// TwinCAT 3 PLC project PLC1
// ProgramVersion: 3.1.4023.0
// libraries:
//   SPT Base Types, * (Beckhoff Automation LLC)
//   SPT Components, * (Beckhoff Automation LLC)
//   SPT Diagnostic, * (Beckhoff Automation LLC)
//   SPT EtherCat, * (Beckhoff Automation LLC)
//   SPT Event Logger, * (Beckhoff Automation LLC)
//   SPT Utilities, * (Beckhoff Automation LLC)
//   Tc2_EtherCAT, * (Beckhoff Automation GmbH)
//   Tc2_Standard, * (Beckhoff Automation GmbH)
//   Tc2_System, * (Beckhoff Automation GmbH)
//   Tc3_EventLogger, * (Beckhoff Automation GmbH)
//   Tc3_Module, * (Beckhoff Automation GmbH)
//   Tc3_PackML_V2, * (Beckhoff Automation GmbH)
//   VisuDialogs, * (System)
//   VisuSymbols,newest,System
// project tree:
//   DUTs/Recipe/NewFolder1/ ST_PullWheelsRecipe.TcDUT, ST_SealerRecipe.TcDUT, ST_UnwindRecipe.TcDUT
//   DUTs/Recipe/ ST_AxisRecipe.TcDUT, ST_ConveyorRecipe.TcDUT, ST_MotionLinxAxisRecipe.TcDUT, ST_StationRecipe.TcDUT, ST_Vision_Volume_Recipe.TcDUT, ST_Diagnostics_Recipe.TcDUT, ST_Gluer_Recipe.TcDUT, ST_DiverterRecipe.TcDUT, ST_Closer_Recipe.TcDUT, ST_LabelerRecipe.TcDUT, ST_OutfeedRecipe.TcDUT, ST_SafetyRecipe.TcDUT
//   DUTs/ ST_Descriptor2.TcDUT (not stored), ST_PackML_Control.TcDUT (not stored), ST_PackML_Control_Simplified.TcDUT (not stored)
//   / GlobalTextList.TcGTLO, MAIN.TcPOU, PlcTask.TcTTO, VisualizationManager.TcVMO (not stored)
//   Machine/Components/Contactor/ FB_Contactor.TcPOU, FB_Contactor_Dual_InOut.TcPOU, FB_Contactor_With_Dual_Feedback.TcPOU, FB_Contactor_With_Single_Feedback.TcPOU, I_Contactor.TcIO, ST_Contactor_Command.TcDUT, ST_Contactor_Config.TcDUT, ST_Contactor_HMI.TcDUT, ST_Contactor_Status.TcDUT
//   Machine/Components/Cylinder/ FB_Cylinder.TcPOU (not stored), I_Cylinder.TcIO (not stored), ST_Cylinder_Command.TcDUT (not stored), ST_Cylinder_Config.TcDUT (not stored), ST_Cylinder_HMI.TcDUT (not stored), ST_Cylinder_Status.TcDUT (not stored)
//   Machine/Components/Drives/ iDM_DriveHealth.TcIO
//   Machine/Components/Drives/Omron/ eDriveStates.TcDUT, eOmronStatus.TcDUT (not stored), FB_BLINKER_PLAY.TcPOU (not stored), FB_Omron_Inv.TcPOU, stOmronDriveMapping.TcDUT
//   Machine/Components/Drives/Omron/Old System/DM_Omron/ DM_Omron_Drive.TcPOU
//   Machine/Components/Drives/Roller Drives/2 Motor Drive/Axis/ FB_Drive_Type_1_Axis.TcPOU, I_Drive_Type_1_Axis.TcIO
//   Machine/Components/Drives/Roller Drives/2 Motor Drive/ FB_Drive_Type_1_Controller.TcPOU, I_Drive_Type_1_Controller.TcIO
//   Machine/Components/ FB_SealBar.TcPOU (not stored)
//   Machine/Components/MotionLinxAI/Axis/ FB_MotionlinxAI_Axis.TcPOU, I_MotionlinxAI_Axis.TcIO, MotionlinxAI_Error_States.TcDUT, MotionlinxAI_Motor_Status.TcDUT, ST_MotionlinxAI_Axis_Command.TcDUT, ST_MotionlinxAI_Axis_Config.TcDUT, ST_MotionlinxAI_Axis_HMI.TcDUT, ST_MotionlinxAI_Axis_Status.TcDUT
//   Machine/Components/MotionLinxAI/Axis/HMI/ ST_MotionlinxAI_Controller_Command.TcDUT, ST_MotionlinxAI_Controller_Config.TcDUT, ST_MotionlinxAI_Controller_HMI.TcDUT, ST_MotionlinxAI_Controller_Status.TcDUT
//   Machine/Components/MotionLinxAI/Controller/ FB_MotionlinxAI_Controller.TcPOU, I_MotionlinxAI_Controller_Sts.TcIO, ST_Controller_Status.TcDUT
//   Machine/Components/MotionLinxAI/ MotionlinxAI_States.TcDUT
//   Machine/Components/Relay/ I_Relay.TcIO, Relay.TcPOU, Relay_Pulse.TcPOU
//   Machine/Components/Robots/ GVL_UR.TcGVL
//   Machine/Components/Robots/UR/ fbUR.TcPOU
//   Machine/Components/Robots/UR/IO-Mapping/Structs/ stUR_EIO_Output_Mapping.TcDUT, stUR_EIO_Safety_Bits_Mapping.TcDUT, UR_Output_Data.TcDUT, UR_Safety_Bits_Data.TcDUT
//   Machine/Components/Vision/Cognex/ FB_A100.TcPOU
//   Machine/EquipmentModules/Conveyors/ FB_Robot_Outfeed_Conveyor_Module.TcPOU, FB_SingleDrive_Conveyor_With_Out_Sensor.TcPOU, FB_SingleDrive_Conveyor_With_Out_Sensor_And_Stopper.TcPOU, FB_Single_Drive_Outfeed_Sensor.TcPOU
//   Machine/EquipmentModules/ FB_Diverter_Module.TcPOU, FB_Station_Module.TcPOU, FB_Labeler_Module.TcPOU, FB_Closer_Gluer_Module.TcPOU, FB_Outfeed_Conveyor_Module_OLD.TcPOU (excluded from build)
//   Machine/EquipmentSubModules/ FB_Diverter_Module001.TcPOU, FB_Gluer_Module.TcPOU, FB_Vision_Volume_SubModule.TcPOU, FB_Vision_Barcode_SubModule.TcPOU, FB_Labeler_SubModule.TcPOU
//   Machine/ FB_Machine.TcPOU, FB_Safety.TcPOU (excluded from build), FB_Systems.TcPOU (excluded from build)
//   Machine/HMI Connections/ FB_ControlSource_HMI.TcPOU (not stored), FB_ControlSource_HMI_Machine.TcPOU
//   Machine/MachineSubModules/ FB_Diagnostics_SubModule.TcPOU, FB_Systems_Module.TcPOU
//   Machine/SafetyModules/ FB_Safety_Module.TcPOU
//   Machine/Templates/ FB_EquipmentModuleTemplate.TcPOU (not stored)
//   Machine/VISUs/VisuOjects/ V_EtherCatMasterComponent.TcVIS, V_MachineModule.TcVIS, V_SafetyModule.TcVIS, V_Module.TcVIS (not stored)
//   Machine/VISUs/ V_Main.TcVIS
// real-time tasks:
//   TASK PlcTask: cycle T#10ms, priority 10, ADS port 350
// motion (NC):
//   TASK NC-Task 1 SAF: cycle T#2ms, priority 4, ADS port 501
//   TASK NC-Task 1 SVB: cycle T#10ms, priority 8, ADS port 511
//   AXIS Unwind (id 4)
//   AXIS Seal (id 5)
//   AXIS Pull 1 (id 6)
//   AXIS Pull 2 (id 7)
// I/O:
//   DEVICE Device 2 (RT-Ethernet Adapter) DO NOT DELETE
//   DEVICE Device 5 (EtherCAT), AmsNetId 192.168.100.70.6.1
//     Box 1 (CU2508) [CU2508 Ethernet Port]
//     Term 2 (EK1100) [EK1100 EtherCAT Coupler (2A E-Bus)]
//       Term 3 (EL1904) [EL1904, 4 Ch. Safety Input 24V, TwinSAFE]
//         modules: Module 1 (FSOES)
//       Term 4 (EL1904) [EL1904, 4 Ch. Safety Input 24V, TwinSAFE]
//         modules: Module 1 (FSOES)
//       Term 5 (EL2904) [EL2904, 4 Ch. Safety Output 24V, 0.5A, TwinSAFE]
//         modules: Module 1 (FSOES), Module 2 (DO)
//       Term 6 (EL6900) [EL6900, TwinSAFE PLC]
//       Term 7 (EL2008) [EL2008 8Ch. Dig. Output 24V, 0.5A]
//       Term 8 (EL1008) [EL1008 8Ch. Dig. Input 24V, 3ms]
//       Term 9 (EL9011) [EL9011 End Terminal]
//     Box 18 (MotionLinx-Ai PLCmode) [MotionLinx-Ai PLCmode FW4.1]
// variable links:
//   PLC1/PLC1 Instance <-> Device 5 (EtherCAT)
//     PlcTask Inputs/MAIN.Machine.Systems_SubModule.Diagnostics.EtherCatMasterX001.EtherCatMaster.AmsNetID <-> InfoData/AmsNetId
//     PlcTask Inputs/MAIN.Machine.Systems_SubModule.Diagnostics.EtherCatMasterX001.EtherCatMaster.CfgSlaveCount <-> InfoData/CfgSlaveCount
//     PlcTask Inputs/MAIN.Machine.Systems_SubModule.Diagnostics.EtherCatMasterX001.EtherCatMaster.ChangeCount <-> InfoData/ChangeCount
//     PlcTask Inputs/MAIN.Machine.Systems_SubModule.Diagnostics.EtherCatMasterX001.EtherCatMaster.DevID <-> InfoData/DevId
//     PlcTask Inputs/MAIN.Machine.Systems_SubModule.Diagnostics.EtherCatMasterX001.EtherCatMaster.DevState <-> Inputs/DevState
//     PlcTask Inputs/MAIN.Machine.Systems_SubModule.Diagnostics.EtherCatMasterX001.EtherCatMaster.SlaveCount <-> Inputs/SlaveCount
//     PlcTask Inputs/MAIN.Machine.Systems_SubModule.Diagnostics.EtherCatMasterX001.FrmXWcState[0] <-> Inputs/Frm0State
//   PLC1/PLC1 Instance <-> Device 5 (EtherCAT)/Box 18 (MotionLinx-Ai PLCmode)
//     PlcTask Inputs/MAIN.Machine.Diverter_MotionlinxAI_Controller.bInputToggle <-> WcState/InputToggle
//     PlcTask Inputs/MAIN.Machine.Diverter_MotionlinxAI_Controller.bWCState <-> WcState/WcState
//     PlcTask Inputs/MAIN.Machine.Diverter_MotionlinxAI_Controller.iSensors <-> Module Inputs/AllSensors
//     PlcTask Inputs/MAIN.Machine.Diverter_MotionlinxAI_Controller.iSysDiagnostics <-> Module Diagnostics/SystemDiagnostic
//     PlcTask Inputs/MAIN.Machine.Station_1.Axis.iDiagnostics <-> Module Diagnostics/DiagnosticLeft
//     PlcTask Inputs/MAIN.Machine.Station_1.Axis.iPosition <-> Module Inputs/PositionLeft
//     PlcTask Inputs/MAIN.Machine.Station_1.Axis.iServoState <-> Module Inputs/ServoStateL
//     PlcTask Inputs/MAIN.Machine.Station_5.Axis.iDiagnostics <-> Module Diagnostics/DiagnosticRight
//     PlcTask Inputs/MAIN.Machine.Station_5.Axis.iPosition <-> Module Inputs/PositionRight
//     PlcTask Inputs/MAIN.Machine.Station_5.Axis.iServoState <-> Module Inputs/ServoStateR
//     PlcTask Outputs/MAIN.Machine.Diverter_MotionlinxAI_Controller.oClearMotorError <-> Servo/Periphery/ClearMotorError
//     PlcTask Outputs/MAIN.Machine.Diverter_MotionlinxAI_Controller.oServoControl <-> Servo/Periphery/ServoCtrl
//     PlcTask Outputs/MAIN.Machine.Diverter_MotionlinxAI_Controller.oSetPin2Out <-> Servo/Periphery/WritePin2Output
//     PlcTask Outputs/MAIN.Machine.Station_1.Axis.oMotorAccel <-> Motor Ramps/AccelLeft
//     PlcTask Outputs/MAIN.Machine.Station_1.Axis.oMotorBrakeMode <-> Motor Setup/BrakeModeLeft
//     PlcTask Outputs/MAIN.Machine.Station_1.Axis.oMotorControl <-> Motor Setup/MDRCtrlLeft
//     PlcTask Outputs/MAIN.Machine.Station_1.Axis.oMotorDecel <-> Motor Ramps/DecelLeft
//     PlcTask Outputs/MAIN.Machine.Station_1.Axis.oMotorSpeed <-> Motor Setup/SpeedLeft
//     PlcTask Outputs/MAIN.Machine.Station_1.Axis.oServoPos <-> Servo/Periphery/ServoLeft
//     PlcTask Outputs/MAIN.Machine.Station_5.Axis.oMotorAccel <-> Motor Ramps/AccelRight
//     PlcTask Outputs/MAIN.Machine.Station_5.Axis.oMotorBrakeMode <-> Motor Setup/BrakeModeRight
//     PlcTask Outputs/MAIN.Machine.Station_5.Axis.oMotorControl <-> Motor Setup/MDRCtrlRight
//     PlcTask Outputs/MAIN.Machine.Station_5.Axis.oMotorDecel <-> Motor Ramps/DecelRight
//     PlcTask Outputs/MAIN.Machine.Station_5.Axis.oMotorSpeed <-> Motor Setup/SpeedRight
//     PlcTask Outputs/MAIN.Machine.Station_5.Axis.oServoPos <-> Servo/Periphery/ServoRight
//   PLC1/PLC1 Instance <-> Device 5 (EtherCAT)/Term 2 (EK1100)/Term 6 (EL6900)
//     PlcTask Inputs/MAIN.Machine.Safety_SubModule.SafetyEstop.InfoData/Diag <-> TwinSAFE Group Info Data/TwinSafeGroup_Estop Info Data/Diag
//     PlcTask Inputs/MAIN.Machine.Safety_SubModule.SafetyEstop.InfoData/State <-> TwinSAFE Group Info Data/TwinSafeGroup_Estop Info Data/State
//     PlcTask Inputs/MAIN.Machine.Safety_SubModule.SafetyGroup_ESTOP.InfoData/Diag <-> Function Block Info Data/TwinSafeGroup_Estop.ESTOP_Circuit.FBEstop1 Info Data/Diag
//     PlcTask Inputs/MAIN.Machine.Safety_SubModule.SafetyGroup_ESTOP.InfoData/State <-> Function Block Info Data/TwinSafeGroup_Estop.ESTOP_Circuit.FBEstop1 Info Data/State
//     PlcTask Inputs/MAIN.Machine.Safety_SubModule.SafetyGroup_IO.InfoData/Diag <-> TwinSAFE Group Info Data/TwinSafeGroup_IO Info Data/Diag
//     PlcTask Inputs/MAIN.Machine.Safety_SubModule.SafetyGroup_IO.InfoData/State <-> TwinSAFE Group Info Data/TwinSafeGroup_IO Info Data/State
//     PlcTask Inputs/MAIN.Machine.Safety_SubModule.SafetyInput.InfoData/Diag <-> Connection Info Data/Message_5 Info Data/Diag
//     PlcTask Inputs/MAIN.Machine.Safety_SubModule.SafetyInput.InfoData/State <-> Connection Info Data/Message_5 Info Data/State
//     PlcTask Inputs/MAIN.Machine.Safety_SubModule.SafetyOutput.InfoData/Diag <-> Connection Info Data/Message_7 Info Data/Diag
//     PlcTask Inputs/MAIN.Machine.Safety_SubModule.SafetyOutput.InfoData/State <-> Connection Info Data/Message_7 Info Data/State
//     PlcTask Outputs/MAIN.Machine.Safety_SubModule.SafetyGroup_ESTOP.Run <-> StandardOutputs/Standard In Var 14
//     PlcTask Outputs/MAIN.Machine.Safety_SubModule.SafetyGroup_IO.Run <-> StandardOutputs/Standard In Var 4
//     PlcTask Outputs/MAIN.Machine.Safety_SubModule.Safty_Reset_Pulse_Out.output <-> StandardOutputs/Standard In Var 12
//     PlcTask Outputs/MAIN.Machine.Safety_SubModule.Safty_Reset_Pulse_Out.output <-> StandardOutputs/Standard In Var 3
//   (this object) <-> Device 5 (EtherCAT)
//     Term 2 (EK1100)/Term 3 (EL1904)/Module 1 (FSOES)/RxPDO/FSOE <-> Term 2 (EK1100)/Term 6 (EL6900)/ConnectionInputs/Message_5 TxPDO
//     Term 2 (EK1100)/Term 5 (EL2904)/Module 1 (FSOES)/RxPDO/FSOE <-> Term 2 (EK1100)/Term 6 (EL6900)/ConnectionInputs/Message_7 TxPDO
//     Term 2 (EK1100)/Term 3 (EL1904)/Module 1 (FSOES)/TxPDO/FSOE <-> Term 2 (EK1100)/Term 6 (EL6900)/ConnectionOutputs/Message_5 RxPDO
//     Term 2 (EK1100)/Term 5 (EL2904)/Module 1 (FSOES)/TxPDO/FSOE <-> Term 2 (EK1100)/Term 6 (EL6900)/ConnectionOutputs/Message_7 RxPDO
//     Term 2 (EK1100)/Term 6 (EL6900)/ConnectionInputs/Message_5 TxPDO <-> Term 2 (EK1100)/Term 3 (EL1904)/Module 1 (FSOES)/RxPDO/FSOE
//     Term 2 (EK1100)/Term 6 (EL6900)/ConnectionInputs/Message_7 TxPDO <-> Term 2 (EK1100)/Term 5 (EL2904)/Module 1 (FSOES)/RxPDO/FSOE
//     Term 2 (EK1100)/Term 6 (EL6900)/ConnectionOutputs/Message_5 RxPDO <-> Term 2 (EK1100)/Term 3 (EL1904)/Module 1 (FSOES)/TxPDO/FSOE
//     Term 2 (EK1100)/Term 6 (EL6900)/ConnectionOutputs/Message_7 RxPDO <-> Term 2 (EK1100)/Term 5 (EL2904)/Module 1 (FSOES)/TxPDO/FSOE

CONFIGURATION PLC1
    RESOURCE PLC ON TwinCAT3
        TASK PlcTask(INTERVAL := T#10ms, PRIORITY := 10);
        PROGRAM MAIN WITH PlcTask : MAIN;
    END_RESOURCE
END_CONFIGURATION

// ---- DUTs/Recipe/NewFolder1/ST_PullWheelsRecipe.TcDUT
TYPE ST_PullWheelsRecipe :
	STRUCT
		Length				: LREAL;
		LeftAxis			: ST_AxisRecipe;
		RightAxis			: ST_AxisRecipe;
		CylinderExtendTime	: LREAL;
		CylinderRetractTime : LREAL;
	END_STRUCT
END_TYPE

// ---- DUTs/Recipe/NewFolder1/ST_SealerRecipe.TcDUT
TYPE ST_SealerRecipe :
	STRUCT
		Axis		   : ST_AxisRecipe;
		Temp		   : LREAL;
		SealTime	   : LREAL;
		OpenPosition   : LREAL;
		ClosedPosition : LREAL;
	END_STRUCT
END_TYPE

// ---- DUTs/Recipe/NewFolder1/ST_UnwindRecipe.TcDUT
TYPE ST_UnwindRecipe :
	STRUCT
		Axis : ST_AxisRecipe;
	END_STRUCT
END_TYPE

// ---- DUTs/Recipe/ST_AxisRecipe.TcDUT
TYPE ST_AxisRecipe :
	STRUCT
		Velocity		: INT;
		Acceleration	: INT;
		Deceleration	: INT;
	//	Speed			: INT;
		MaxVelocity		: INT;
	END_STRUCT
END_TYPE

// ---- DUTs/Recipe/ST_ConveyorRecipe.TcDUT
TYPE ST_ConveyorRecipe :
	STRUCT
		Axis : ST_MotionLinxAxisRecipe;
		
	END_STRUCT
END_TYPE

// ---- DUTs/Recipe/ST_MotionLinxAxisRecipe.TcDUT
TYPE ST_MotionLinxAxisRecipe :
	STRUCT
		Velocity		: INT;
		Acceleration	: INT;
		Deceleration	: INT;	
		MaxSpeed		:UINT;
	END_STRUCT
END_TYPE

// ---- DUTs/Recipe/ST_StationRecipe.TcDUT
TYPE ST_StationRecipe :
STRUCT

		Axis			: ST_AxisRecipe;
		//	Travel Time ??
END_STRUCT
END_TYPE

// ---- DUTs/Recipe/ST_Vision_Volume_Recipe.TcDUT
TYPE ST_Vision_Volume_Recipe :
	STRUCT
		Length				: LREAL;
//		LeftAxis			: ST_AxisRecipe;
//		RightAxis			: ST_AxisRecipe;
		CylinderExtendTime	: LREAL;
		CylinderRetractTime : LREAL;
	END_STRUCT
END_TYPE

// ---- DUTs/Recipe/ST_Diagnostics_Recipe.TcDUT
TYPE ST_Diagnostics_Recipe :
	STRUCT
		Length				: LREAL;
//		LeftAxis			: ST_AxisRecipe;
//		RightAxis			: ST_AxisRecipe;
		CylinderExtendTime	: LREAL;
		CylinderRetractTime : LREAL;
	END_STRUCT
END_TYPE

// ---- DUTs/Recipe/ST_Gluer_Recipe.TcDUT
TYPE ST_Gluer_Recipe :
	STRUCT
		Length				: LREAL;
			// Data
		SetTemperature	   : LREAL;
		Trigger_Delay		: TIME;	
//		LeftAxis			: ST_AxisRecipe;
//		RightAxis			: ST_AxisRecipe;
		CylinderExtendTime	: LREAL;
		CylinderRetractTime : LREAL;
	END_STRUCT
END_TYPE

// ---- DUTs/Recipe/ST_DiverterRecipe.TcDUT
TYPE ST_DiverterRecipe :
	STRUCT
		Length				: LREAL;
//		LeftAxis			: ST_AxisRecipe;
//		RightAxis			: ST_AxisRecipe;
		CylinderExtendTime	: LREAL;
		CylinderRetractTime : LREAL;
	END_STRUCT
END_TYPE

// ---- DUTs/Recipe/ST_Closer_Recipe.TcDUT
TYPE ST_Closer_Recipe :
	STRUCT
		Length				: LREAL;
//		LeftAxis			: ST_AxisRecipe;
//		RightAxis			: ST_AxisRecipe;
		CylinderExtendTime	: LREAL;
		CylinderRetractTime : LREAL;
	END_STRUCT
END_TYPE

// ---- DUTs/Recipe/ST_LabelerRecipe.TcDUT
TYPE ST_LabelerRecipe :
	STRUCT
		Length				: LREAL;
//		LeftAxis			: ST_AxisRecipe;
//		RightAxis			: ST_AxisRecipe;
		CylinderExtendTime	: LREAL;
		CylinderRetractTime : LREAL;
	END_STRUCT
END_TYPE

// ---- DUTs/Recipe/ST_OutfeedRecipe.TcDUT
TYPE ST_OutfeedRecipe :
	STRUCT
		Length				: LREAL;
//		LeftAxis			: ST_AxisRecipe;
//		RightAxis			: ST_AxisRecipe;
		CylinderExtendTime	: LREAL;
		CylinderRetractTime : LREAL;
	END_STRUCT
END_TYPE

// ---- DUTs/Recipe/ST_SafetyRecipe.TcDUT
TYPE ST_SafetyRecipe :
	STRUCT
		Axis : ST_AxisRecipe;
	END_STRUCT
END_TYPE

// ---- Machine/Components/Contactor/ST_Contactor_Command.TcDUT
TYPE ST_Contactor_Command :
    STRUCT
        Extend  : BOOL;
        Retract : BOOL;
    END_STRUCT
END_TYPE

// ---- Machine/Components/Contactor/ST_Contactor_Config.TcDUT
TYPE ST_Contactor_Config :
    STRUCT
        ExtendTime  : LREAL;
        RetractTime : LREAL;
    END_STRUCT
END_TYPE

// ---- Machine/Components/Contactor/ST_Contactor_HMI.TcDUT
TYPE ST_Contactor_HMI :
    STRUCT
        Config  : ST_Contactor_Config;
        Command : ST_Contactor_Command;
        Status  : ST_Contactor_Status;
    END_STRUCT
END_TYPE

// ---- Machine/Components/Contactor/ST_Contactor_Status.TcDUT
TYPE ST_Contactor_Status :
    STRUCT
        Extended   : BOOL;
        Retracted  : BOOL;
        Extending  : BOOL;
        Retracting : BOOL;
    END_STRUCT
END_TYPE

// ---- Machine/Components/Drives/Omron/eDriveStates.TcDUT
{attribute 'qualified_only'}
{attribute 'strict'}
{attribute 'to_string'}
TYPE eDriveStates :
(
	FAULT := 0,
	FAULT_STOPPING,
 	AWAITING_RESET,
	RESET,
	DISABLED,
	STOPPED,	
	STOPPING,
	STARTING,
	RUNNING
);
END_TYPE

// ---- Machine/Components/Drives/Omron/stOmronDriveMapping.TcDUT
TYPE stOmronDriveMapping :
STRUCT
	
	//Inputs
	inInputTerminal AT %I* : UINT;
	inMotorCurrent AT %I* : UINT;	
	inFinTemp AT %I* : UINT;
	inStatus AT %I* : UINT;
	inOutputFrequency AT %I* : UINT;	
	ibWcState AT %I* : BOOL;
	
	inPulse AT %I* : UINT; // not used 

	inErrorCode AT %I* : UINT;  // NOT used 
	inErrorSubCode AT %I* : UINT; // not used 
	inSTOActive  	AT %I* : BOOL; // not mapped 
		
	//Outputs
	onCommand AT %Q* : UINT;
	onFrequencyRef AT %Q* : UINT;
	onAccelTime AT %Q* : UINT;
	onDecelTime AT %Q* : UINT;
			
END_STRUCT
END_TYPE

// ---- Machine/Components/MotionLinxAI/Axis/HMI/ST_MotionlinxAI_Controller_Command.TcDUT
TYPE ST_MotionlinxAI_Controller_Command :
	STRUCT
		Extend	: BOOL;
		Retract : BOOL;
	END_STRUCT
END_TYPE

// ---- Machine/Components/MotionLinxAI/Axis/HMI/ST_MotionlinxAI_Controller_Config.TcDUT
TYPE ST_MotionlinxAI_Controller_Config :
	STRUCT
		ExtendTime	: LREAL;
		RetractTime : LREAL;
	END_STRUCT
END_TYPE

// ---- Machine/Components/MotionLinxAI/Axis/HMI/ST_MotionlinxAI_Controller_HMI.TcDUT
TYPE ST_MotionlinxAI_Controller_HMI :
	STRUCT
		Config	: ST_MotionlinxAI_Controller_Config;
		Command : ST_MotionlinxAI_Controller_Command;
		Status	: ST_MotionlinxAI_Controller_Status;
	END_STRUCT
END_TYPE

// ---- Machine/Components/MotionLinxAI/Axis/HMI/ST_MotionlinxAI_Controller_Status.TcDUT
TYPE ST_MotionlinxAI_Controller_Status :
	STRUCT
		Extended   : BOOL;
		Retracted  : BOOL;
		Extending  : BOOL;
		Retracting : BOOL;
	END_STRUCT
END_TYPE

// ---- Machine/Components/MotionLinxAI/Axis/MotionlinxAI_Error_States.TcDUT
{attribute 'qualified_only'}
{attribute 'strict'}
TYPE MotionlinxAI_Error_States :
(
	
	NO_ERROR,
	MOTOR_SPEED_HI,
	MOTOR_SPEED_LO,
	MOTOR_BOARD_OVERHEAT,
	MOTOR_OVERVOLTAGE,
	MOTOR_UNDERVOLTAGE,
	MOTOR_OVERHEATED,
	MOTOR_MAX_TORQUE,
	MOTOR_SHORT_CIRCUIT,
	MOTOR_NOT_CONNECTED,
	MOTOR_OVERLOADED,
	MOTOR_STALLED,
	MOTOR_HALL_SENSOR
);
END_TYPE

// ---- Machine/Components/MotionLinxAI/Axis/MotionlinxAI_Motor_Status.TcDUT
{attribute 'qualified_only'}
TYPE MotionlinxAI_Motor_Status :
(
	MOTOR_NOT_RUNNING_BRAKED := 0 ,
	MOTOR_NOT_RUNNING_UNBRAKED,
	MOTOR_RUNNING_CCW,
	MOTOR_RUNNING_CW

);
END_TYPE

// ---- Machine/Components/MotionLinxAI/Axis/ST_MotionlinxAI_Axis_Command.TcDUT
TYPE ST_MotionlinxAI_Axis_Command :
	STRUCT
		Extend	: BOOL;
		Retract : BOOL;
	END_STRUCT
END_TYPE

// ---- Machine/Components/MotionLinxAI/Axis/ST_MotionlinxAI_Axis_Config.TcDUT
TYPE ST_MotionlinxAI_Axis_Config :
	STRUCT
		ExtendTime	: LREAL;
		RetractTime : LREAL;
	END_STRUCT
END_TYPE

// ---- Machine/Components/MotionLinxAI/Axis/ST_MotionlinxAI_Axis_HMI.TcDUT
TYPE ST_MotionlinxAI_Axis_HMI :
	STRUCT
		Config	: ST_MotionlinxAI_Axis_Config;
		Command : ST_MotionlinxAI_Axis_Command;
		Status	: ST_MotionlinxAI_Axis_Status;
	END_STRUCT
END_TYPE

// ---- Machine/Components/MotionLinxAI/Axis/ST_MotionlinxAI_Axis_Status.TcDUT
TYPE ST_MotionlinxAI_Axis_Status :
	STRUCT
		Extended   : BOOL;
		Retracted  : BOOL;
		Extending  : BOOL;
		Retracting : BOOL;
	END_STRUCT
END_TYPE

// ---- Machine/Components/MotionLinxAI/Controller/ST_Controller_Status.TcDUT
TYPE ST_Controller_Status :
STRUCT
	HasFault : BOOL;
	bEnabled : BOOL;
	Sensors : INT;
END_STRUCT
END_TYPE

// ---- Machine/Components/MotionLinxAI/MotionlinxAI_States.TcDUT
{attribute 'qualified_only'}
{attribute 'strict'}
TYPE MotionlinxAI_States :
(
	ERROR := 0,
	HOMING,
	STOPPED,
	RUNNING
);
END_TYPE

// ---- Machine/Components/Robots/UR/IO-Mapping/Structs/stUR_EIO_Output_Mapping.TcDUT
TYPE stUR_EIO_Output_Mapping :
STRUCT
	obBrakeRelease		:	BIT;
	{attribute 'hide'}
	Reserved_UR_1  : BIT;
	{attribute 'hide'}
	Reserved_UR_2  : BIT;
	{attribute 'hide'}
	Reserved_UR_3  : BIT;
	{attribute 'hide'}
	Reserved_UR_4  : BIT;
	{attribute 'hide'}
	Reserved_UR_5  : BIT;
	{attribute 'hide'}
	Reserved_UR_6  : BIT;
	{attribute 'hide'}
	Reserved_UR_7  : BIT;
	{attribute 'hide'}
	Reserved_UR_8  : BIT;
	{attribute 'hide'}
	Reserved_UR_9  : BIT;
	{attribute 'hide'}
	Reserved_UR_10  : BIT;
	{attribute 'hide'}
	Reserved_UR_11  : BIT;
	{attribute 'hide'}
	Reserved_UR_12  : BIT;
	{attribute 'hide'}
	Reserved_UR_13  : BIT;
	{attribute 'hide'}
	Reserved_UR_14  : BIT;
	{attribute 'hide'}
	Reserved_UR_15  : BIT;
	{attribute 'hide'}
	Reserved_UR_16  : BIT;
	{attribute 'hide'}
	Reserved_UR_17  : BIT;
	{attribute 'hide'}
	Reserved_UR_18  : BIT;
	{attribute 'hide'}
	Reserved_UR_19  : BIT;
	{attribute 'hide'}
	Reserved_UR_20  : BIT;
	{attribute 'hide'}
	Reserved_UR_21  : BIT;
	{attribute 'hide'}
	Reserved_UR_22  : BIT;
	{attribute 'hide'}
	Reserved_UR_23  : BIT;
	{attribute 'hide'}
	Reserved_UR_24  : BIT;
	{attribute 'hide'}
	Reserved_UR_25  : BIT;
	{attribute 'hide'}
	Reserved_UR_26  : BIT;
	{attribute 'hide'}
	Reserved_UR_27  : BIT;
	{attribute 'hide'}
	Reserved_UR_28  : BIT;
	{attribute 'hide'}
	Reserved_UR_29  : BIT;
	{attribute 'hide'}
	Reserved_UR_30  : BIT;
	{attribute 'hide'}
	Reserved_UR_31  : BIT;
END_STRUCT
END_TYPE

// ---- Machine/Components/Robots/UR/IO-Mapping/Structs/stUR_EIO_Safety_Bits_Mapping.TcDUT
TYPE stUR_EIO_Safety_Bits_Mapping :
STRUCT
	ibNormalMode   : BIT;
	ibReducedMode  : BIT;
	{attribute 'hide'}
	Reserved_UR_2  : BIT;
	{attribute 'hide'}
	Reserved_UR_3  : BIT;
	{attribute 'hide'}
	Reserved_UR_4  : BIT;
	{attribute 'hide'}
	Reserved_UR_5  : BIT;
	{attribute 'hide'}
	Reserved_UR_6  : BIT;
	{attribute 'hide'}
	Reserved_UR_7  : BIT;
	{attribute 'hide'}
	Reserved_UR_8  : BIT;
	{attribute 'hide'}
	Reserved_UR_9  : BIT;
	{attribute 'hide'}
	Reserved_UR_10  : BIT;
	{attribute 'hide'}
	Reserved_UR_11  : BIT;
	{attribute 'hide'}
	Reserved_UR_12  : BIT;
	{attribute 'hide'}
	Reserved_UR_13  : BIT;
	{attribute 'hide'}
	Reserved_UR_14  : BIT;
	{attribute 'hide'}
	Reserved_UR_15  : BIT;
	{attribute 'hide'}
	Reserved_UR_16  : BIT;
	{attribute 'hide'}
	Reserved_UR_17  : BIT;
	{attribute 'hide'}
	Reserved_UR_18  : BIT;
	{attribute 'hide'}
	Reserved_UR_19  : BIT;
	{attribute 'hide'}
	Reserved_UR_20  : BIT;
	{attribute 'hide'}
	Reserved_UR_21  : BIT;
	{attribute 'hide'}
	Reserved_UR_22  : BIT;
	{attribute 'hide'}
	Reserved_UR_23  : BIT;
	{attribute 'hide'}
	Reserved_UR_24  : BIT;
	{attribute 'hide'}
	Reserved_UR_25  : BIT;
	{attribute 'hide'}
	Reserved_UR_26  : BIT;
	{attribute 'hide'}
	Reserved_UR_27  : BIT;
	{attribute 'hide'}
	Reserved_UR_28  : BIT;
	{attribute 'hide'}
	Reserved_UR_29  : BIT;
	{attribute 'hide'}
	Reserved_UR_30  : BIT;
	{attribute 'hide'}
	Reserved_UR_31  : BIT;

END_STRUCT
END_TYPE

// ---- Machine/Components/Robots/UR/IO-Mapping/Structs/UR_Output_Data.TcDUT
TYPE UR_Output_Data :
UNION
	odwURRawOutputData : DWORD;
	data : stUR_EIO_Output_Mapping;
END_UNION
END_TYPE

// ---- Machine/Components/Robots/UR/IO-Mapping/Structs/UR_Safety_Bits_Data.TcDUT
TYPE UR_Safety_Bits_Data :
UNION
	idwURRawInputData : DWORD;
	data : stUR_EIO_Safety_Bits_Mapping;
END_UNION
END_TYPE

// ---- Machine/Components/Robots/GVL_UR.TcGVL
{attribute 'qualified_only'}
VAR_GLOBAL
	UR		 : fbUR;

	ibURPowered				AT %I* : BOOL;
	obURPowerOn				AT %Q* : BOOL;
	
	ibURProtectiveStopOK		AT %I* : BOOL;

END_VAR

// ---- Machine/Components/Contactor/I_Contactor.TcIO
INTERFACE I_Contactor

METHOD Extend
VAR_INPUT
END_VAR
END_METHOD

PROPERTY Extended : BOOL
GET
END_GET
END_PROPERTY

PROPERTY ExtendTime : LREAL
GET
END_GET
SET
END_SET
END_PROPERTY

METHOD Retract
VAR_INPUT
END_VAR
END_METHOD

PROPERTY Retracted : BOOL
GET
END_GET
END_PROPERTY

PROPERTY RetractTime : LREAL
GET
END_GET
SET
END_SET
END_PROPERTY

END_INTERFACE

// ---- Machine/Components/Drives/iDM_DriveHealth.TcIO
INTERFACE iDM_DriveHealth

METHOD Disable : BOOL
VAR_INPUT
END_VAR
END_METHOD

METHOD Enable : BOOL
VAR_INPUT
END_VAR
END_METHOD

PROPERTY FaultLocation : STRING(50)
GET
END_GET
END_PROPERTY

PROPERTY HasFault : BOOL
GET
END_GET
END_PROPERTY

PROPERTY IsReady : BOOL
GET
END_GET
END_PROPERTY

PROPERTY IsRunning : BOOL
GET
END_GET
END_PROPERTY

METHOD Reset : BOOL
VAR_INPUT
END_VAR
END_METHOD

END_INTERFACE

// ---- Machine/Components/Drives/Roller Drives/2 Motor Drive/Axis/I_Drive_Type_1_Axis.TcIO
INTERFACE I_Drive_Type_1_Axis

METHOD Drive : BOOL
VAR_INPUT
END_VAR
END_METHOD

PROPERTY Position : real
GET
END_GET
SET
END_SET
END_PROPERTY

END_INTERFACE

// ---- Machine/Components/Drives/Roller Drives/2 Motor Drive/I_Drive_Type_1_Controller.TcIO
INTERFACE I_Drive_Type_1_Controller

END_INTERFACE

// ---- Machine/Components/MotionLinxAI/Axis/I_MotionlinxAI_Axis.TcIO
INTERFACE I_MotionlinxAI_Axis

PROPERTY HasFault : BOOL
GET
END_GET
END_PROPERTY

PROPERTY IsEnabled : BOOL
GET
END_GET
END_PROPERTY

PROPERTY IsReady : BOOL
GET
END_GET
END_PROPERTY

END_INTERFACE

// ---- Machine/Components/MotionLinxAI/Controller/I_MotionlinxAI_Controller_Sts.TcIO
INTERFACE I_MotionlinxAI_Controller_Sts

METHOD Disable : BOOL
(*BRAKING MODES:
	0 : NORMAL - HOLDS IN PLACE BY SHORTING WINDINGS
	1 : FREE - NOT HELD IN PLACE
	2 : SERVO - MAINTAINS POSITION BASED ON HALLS EFFECT SENSOR*)
END_METHOD

PROPERTY HasFault : BOOL
GET
END_GET
END_PROPERTY

PROPERTY Sensors : int
GET
END_GET
END_PROPERTY

END_INTERFACE

// ---- Machine/Components/Relay/I_Relay.TcIO
INTERFACE I_Relay

PROPERTY OFF : BOOL
GET
END_GET
END_PROPERTY

PROPERTY ON : Bool
GET
END_GET
END_PROPERTY

METHOD PUBLIC SwitchOff
VAR_INPUT
END_VAR
END_METHOD

METHOD PUBLIC SwitchOn
VAR_INPUT
END_VAR
END_METHOD

END_INTERFACE

// ---- MAIN.TcPOU
PROGRAM MAIN
VAR
	ControlSource_HMI : FB_ControlSource_HMI_Machine;
	
//	Safety		: FB_Safety			:= (Name := 'Safety', DisableSubModuleModeChange	:= TRUE, LogStateChanges	:= TRUE );
//	Systems	  	: FB_Systems := (Name := 'Machine Systems');
	Machine		: FB_Machine := (Name := 'Box Closer Labeler');
	InitComplete	  : BOOL;

	//Debug testing Recipe manager
	Value1 : INT;
	Value2 : INT;
END_VAR

CyclicLogic();
//Did you update??

METHOD CyclicLogic
VAR_INPUT
END_VAR
IF NOT InitComplete THEN
	InitComplete := Initialize();
	RETURN;
END_IF

//Machine support HMI & Production Monitor
ControlSource_HMI.CyclicLogic();

//Safety
//Safety.CyclicLogic();

//Machine Systems 	- Communications, maintenance
//Systems.CyclicLogic();


//Machine Cyclic Logic
Machine.CyclicLogic();
END_METHOD

METHOD Initialize : BOOL
VAR_INPUT
END_VAR
//Top level machine initialization should happen here, in the main initialization method. Each subsequent "layer" of modules will be named within their respective "parent" intialize method
_AppInfo.KeepOutputsOnBP := TRUE;
IF NOT ControlSource_HMI.Registered THEN
	Machine.RegisterExternalController(ControlSource_HMI);
END_IF

ControlSource_HMI.CyclicLogic();
Initialize := TRUE;
END_METHOD

END_PROGRAM

// ---- Machine/HMI Connections/FB_ControlSource_HMI_Machine.TcPOU
FUNCTION_BLOCK FB_ControlSource_HMI_Machine EXTENDS FB_ControlSource_HMI
VAR_INPUT
END_VAR

VAR_OUTPUT
END_VAR

VAR
END_VAR

METHOD CyclicLogic
VAR_INPUT
END_VAR
SUPER^.CyclicLogic();

//Change the start permissive for the Machine 
MainPMLControl_Simplified.StartPermissive := MainPMLControl_Standard.CurrentState = Tc3_PackML_V2.E_PMLState.ePMLState_Idle OR (MainPMLControl_Standard.CurrentState = Tc3_PackML_V2.E_PMLState.ePMLState_Held AND MAIN.Machine.Station_1.CurrentState = E_PMLState.ePMLState_Idle);
//MainPMLControl_Simplified.StartPermissive := MainPMLControl_Standard.CurrentState = Tc3_PackML_V2.E_PMLState.ePMLState_Idle OR (MainPMLControl_Standard.CurrentState = Tc3_PackML_V2.E_PMLState.ePMLState_Held AND MAIN.VFFSDemo.Unwind.CurrentState = E_PMLState.ePMLState_Idle);
END_METHOD

END_FUNCTION_BLOCK

// ---- Machine/FB_Machine.TcPOU
FUNCTION_BLOCK FB_Machine EXTENDS FB_PackML_BaseModule // IMPLEMENTS I_ControlsProductionRate
VAR
	
//	//FB Called  for this machine
//	Diverter_Controller_1	:FB_Drive_Type_1_Controller := (Name := 'Diverter_Controller_1');

	// Components
//	Buffer_1_Outfeed_Sensor :FB_DigitalSensor		:= (Name := 'Sensor', DebounceMode := E_DebounceMode.SimpleFlickerFilter, DebounceTime := T#250MS, Inverted    := FALSE, SimulationInput:= FALSE, SimulationMode := E_SensorSimulationMode.InputDriven) ;
	
	// Sub Modules
	//Safety
	Safety_SubModule			: FB_Safety_Module			:= (Name := 'Safety', LogStateChanges := TRUE);
	
	//Systems
	Systems_SubModule			: FB_Systems_Module	:= (Name := 'Systems', LogStateChanges := TRUE);

	
	Station_1		: FB_Station_Module:= (Name := 'Product Infeed', LogStateChanges := TRUE);
	Station_2		: FB_Station_Module:= (Name := 'Station_2', LogStateChanges := TRUE);
	Station_3		: FB_Station_Module:= (Name := 'Station_3', LogStateChanges := TRUE);
	Station_4		: FB_Station_Module:= (Name := 'Station_4', LogStateChanges := TRUE);
	Station_5			: FB_Station_Module:= (Name := 'Robot Outfeed Station', LogStateChanges := TRUE);
	Station_6		: FB_Station_Module:= (Name := 'UR Robot Station', LogStateChanges := TRUE);
//	Outfeed			: FB_Robot_Outfeed_Conveyor_Module:= (Name := 'Robot Outfeed Station', LogStateChanges := TRUE);
	

	//Initial List of Components
	ipComponents_Init : ARRAY[1..Parameters_PackML_Base.MAX_NO_OF_COMPONENTS] OF I_ComponentBase := [];
	
	//FB Called  for this machine
	Diverter_MotionlinxAI_Controller	:FB_MotionlinxAI_Controller	:= (Name := 'Diverter Drives');
	Diverter_MotionlinxAI_Controller_Sensors	: I_MotionlinxAI_Controller_Sts;
	

	//Alarms for this module
	MachineAlarms : ARRAY[1..MACHINE_ALARM_COUNT] OF FB_TcAlarm;

	//Current Recipe Name
	CurrentRecipeName : STRING;

	//Get Data From PackML? Else RecipeManager is running
	DataFromPackML : BOOL := TRUE;
	Externam_Machine	:I_PackML_ExternalController;

	//Data 
	sealTimeStart : ULINT;
	sealTimeEnd	  : ULINT;
	sealingTime	  : LREAL;
	sealTrig	  : R_TRIG;
	pullTimeStart : ULINT;
	pullTimeEnd	  : ULINT;
	pullingTime	  : LREAL;
	pulltrig	  : R_TRIG;
	partTimeStart : ULINT;
	partTimeEnd	  : ULINT;
	partTime	  : LREAL;
	parts		  : DINT;
	product		  : DINT;

	//Pack Tags for System
	{attribute 'OPC.UA.DA' := '1'}
	_PackTags : ST_PackMLv30Ext; //ST_PackMLv30 is obsolete in Tc3_PackML_V2
END_VAR

VAR CONSTANT
	//PackTag parameter IDs
	LENGTH		   : INT := 1;
	SEALTEMP	   : INT := 2;
	SEALTIME	   : INT := 3;
	PULLWHEELS_VEL : INT := 4;
	PULLWHEELS_ACC : INT := 5;
	SEALER_VEL	   : INT := 6;
	SEALER_ACC	   : INT := 7;
	UNWIND_VEL	   : INT := 8;
	UNWIND_ACC	   : INT := 9;
	OPEN_POS	   : INT := 10;
	CLOSED_POS	   : INT := 11;

	//Alarm count constant
	MACHINE_ALARM_COUNT : INT := 6;
END_VAR

// Simulation variables
VAR
	EstopInput	: BOOL;
	LowAirInput : BOOL;
	ErrorInput	: BOOL;
	WarnInput	: BOOL;
	InfoInput	: BOOL;
END_VAR

(*







*)

METHOD PROTECTED Completing
VAR_INPUT
END_VAR
CASE _CurrentMode OF
	//=================================PRODUCTION MODE==================================
	E_PMLUnitMode.ePMLUnitMode_Production:
		StateComplete();

	E_PMLUnitMode.ePMLUnitMode_Maintenance, E_PMLUnitMode.ePMLUnitMode_Manual:
		SUPER^.Completing();
END_CASE
END_METHOD

METHOD PROTECTED CreateEvents
VAR_INPUT
END_VAR
// Add your event creation here
F_CreateAllEventsInClass(Alarms		:= MachineAlarms,
						 ClassSize	:= SIZEOF(TC_Events.DemoSystem),
						 pInitEvent := ADR(TC_EVENTS.DemoSystem.InitReferenceEvent),
						 Prefix		:= Name);

// Super call to base
SUPER^.CreateEvents();
END_METHOD

METHOD CyclicLogic
VAR_INPUT
END_VAR
IF NOT _InitComplete THEN
	_InitComplete := Initialize();
	RETURN;
END_IF

SUPER^.CyclicLogic();

// Fill in the PackTags for the machine output
_PackTags.Status.StateCurrent	 := _CurrentState;
_PackTags.Status.UnitModeCurrent := _CurrentMode;
UpdateModeTimers();

//Call any locally generated FBs
//Diverter_Controller_1.CyclicLogic();
Station_1.Controller_Sts	:= Diverter_MotionlinxAI_Controller.Controller_Status;
Station_5.Controller_Sts	:= Diverter_MotionlinxAI_Controller.Controller_Status;


//This is just to simulate some IO for alarms
//CyclicLogic_Simulation();
END_METHOD

METHOD CyclicLogic_Simulation
VAR_INPUT
END_VAR

VAR_INST
END_VAR
(*	
This is just for testing. Real hardware can be setup in other places
Here the alarms will raise and clear on its own if the input changes	
*)
IF EstopInput AND NOT MachineAlarms[E_DemoSystem.EmergencyStop].bRaised THEN
	RaiseAlarm2Args(MachineAlarms[E_DemoSystem.EmergencyStop], '', '');
ELSIF NOT EstopInput AND MachineAlarms[E_DemoSystem.EmergencyStop].bRaised THEN
	MachineAlarms[E_DemoSystem.EmergencyStop].Clear(0, 0);
END_IF

IF LowAirInput AND NOT MachineAlarms[E_DemoSystem.LowAir].bRaised THEN
	RaiseAlarm2Args(MachineAlarms[E_DemoSystem.LowAir], '', '');
ELSIF NOT LowAirInput AND MachineAlarms[E_DemoSystem.LowAir].bRaised THEN
	MachineAlarms[E_DemoSystem.LowAir].Clear(0, 0);
END_IF

//Generic Alarms for Testing
IF ErrorInput AND NOT MachineAlarms[E_DemoSystem.AlarmMessage].bRaised THEN
	RaiseAlarm2Args(MachineAlarms[E_DemoSystem.AlarmMessage], '', '');
ELSIF NOT ErrorInput AND MachineAlarms[E_DemoSystem.AlarmMessage].bRaised THEN
	MachineAlarms[E_DemoSystem.AlarmMessage].Clear(0, 0);
END_IF

IF WarnInput AND NOT MachineAlarms[E_DemoSystem.WarnMessage].bRaised THEN
	RaiseAlarm2Args(MachineAlarms[E_DemoSystem.WarnMessage], '', '');
ELSIF NOT WarnInput AND MachineAlarms[E_DemoSystem.WarnMessage].bRaised THEN
	MachineAlarms[E_DemoSystem.WarnMessage].Clear(0, 0);
END_IF

IF InfoInput AND NOT MachineAlarms[E_DemoSystem.InfoMessage].bRaised THEN
	RaiseAlarm2Args(MachineAlarms[E_DemoSystem.InfoMessage], '', '');
ELSIF NOT InfoInput AND MachineAlarms[E_DemoSystem.InfoMessage].bRaised THEN
	MachineAlarms[E_DemoSystem.InfoMessage].Clear(0, 0);
END_IF
END_METHOD

METHOD PROTECTED FINAL Execute
VAR_INPUT
END_VAR
CASE _CurrentMode OF
	//=================================PRODUCTION MODE==================================
	E_PMLUnitMode.ePMLUnitMode_Production:
		(* Run the sequence to make products 
		 Unwind Runs Slowly 
		 Pull Wheels Run 
		 Jaws Seal, and Repeat until production reached*)
		sealTrig(CLK := SequenceState = 10);
		IF sealTrig.Q THEN
			partTimeStart := F_GetActualDcTime64();
			sealTimeStart := partTimeStart;
		END_IF

		pulltrig(CLK := SequenceState = 20);
		IF pulltrig.Q THEN
			pullTimeStart := F_GetActualDcTime64();
		END_IF
//		Station_1.ChangeState(E_PMLCommand.ePMLCommand_Start);
		
//ACTION Depending on how you want control, the Station logic can be programmed to stop the conveyor when the trigger occurs
//	and just monitor/control stated here		
//		IF THIS^.Sealer.sealbar.InTempRange THEN
			CASE SequenceState OF
				0: //Started
					Station_5.ChangeState(E_PMLCommand.ePMLCommand_Start);
					IF Station_5.CurrentState = E_PMLState.ePMLState_Execute THEN
						SequenceState := SequenceState + 10;
					END_IF


				10:	//
					IF Station_5.OutFeed_Sensor.Active THEN
						Station_5.ChangeState(E_PMLCommand.ePMLCommand_Stop);
						SequenceState := SequenceState + 10;
					END_IF
				
				20:
					IF Station_5.CurrentState = E_PMLState.ePMLState_Stopped THEN
						SequenceState := SequenceState + 10;
					END_IF


(*
				0: //Started
					Station_1.ChangeState(E_PMLCommand.ePMLCommand_Start);
					IF Station_1.CurrentState = E_PMLState.ePMLState_Execute THEN
						SequenceState := SequenceState + 10;
					END_IF


				10:	//
					IF Station_1.OutFeed_Sensor.Active THEN
						Station_1.ChangeState(E_PMLCommand.ePMLCommand_Stop);
						SequenceState := SequenceState + 10;
					END_IF
				
				20:
					IF Station_1.CurrentState = E_PMLState.ePMLState_Stopped THEN
						SequenceState := SequenceState + 10;
					END_IF



*)








//				10: // SEAL First
//					Sealer.ChangeState(E_PMLCommand.ePMLCommand_Start);
//					IF Sealer.CurrentState = E_PMLState.ePMLState_Complete THEN
//						Sealer.ChangeState(E_PMLCommand.ePMLCommand_Reset);
//						SequenceState := SequenceState + 10;
//						SealTimeEnd	  := F_GetActualDcTime64();
//						sealingTime	  := ULINT_TO_LREAL(sealtimeEnd - sealTimeStart) * 1E-9;
//					END_IF

//				20: // Run Pullwheels
//					PullWheels.ChangeState(E_PMLCommand.ePMLCommand_Start);
//					IF PullWheels.CurrentState = E_PMLState.ePMLState_Complete THEN
//						partTimeEnd	  := F_GetActualDcTime64();
//						parts		  := parts + 1;
//						SequenceState := 10;
//						PullWheels.ChangeState(E_PMLCommand.ePMLCommand_Reset);
//						pullTimeEnd := F_GetActualDcTime64();
//						pullingTime := ULINT_TO_LREAL(pullTimeEnd - pullTimeStart) * 1E-9;
//					END_IF
			END_CASE
//		ELSE
//			ChangeState(E_PMLCommand.ePMLCommand_Suspend);
//		END_IF

	//=================================MAINTENANCE MODE==================================	
	E_PMLUnitMode.ePMLUnitMode_Maintenance:
		;

	//=================================MANUAL MODE==================================
	E_PMLUnitMode.ePMLUnitMode_Manual:
		;
END_CASE
END_METHOD

METHOD PROTECTED Held
VAR_INPUT
END_VAR
END_METHOD

METHOD PROTECTED HMIPermissions
VAR_INPUT
END_VAR
//General Mode Based Monitoring and handling of HMI control
CASE _CurrentMode OF
	E_PMLUnitMode.ePMLUnitMode_Production:
		CASE _CurrentState OF
			E_PMLState.ePMLState_Stopped:
				AllowHMIControl(ThisModuleOnly := TRUE); //Allow control for recovery
			E_PMLState.ePMLState_Idle:
				//BlockHMIControl();
				AllowHMIControl(ThisModuleOnly := TRUE); //Allow control for recovery
			E_PMLState.ePMLState_Suspended:
				BlockHMIControl();

			E_PMLState.ePMLState_Execute:
				 //BlockHMIControl();
				AllowHMIControl(ThisModuleOnly := TRUE); //Allow control for recovery

			E_PMLState.ePMLState_Aborted:
				AllowHMIControl(ThisModuleOnly := TRUE); //Allow control for recovery
			E_PMLState.ePMLState_Held:
				AllowHMIControl(ThisModuleOnly := TRUE); //Allow control for recovery
			E_PMLState.ePMLState_Complete:
				BlockHMIControl();
		END_CASE

	//AllowHMIControl(ThisModuleOnly := FALSE);
	E_PMLUnitMode.ePMLUnitMode_Manual:
		AllowHMIControl(ThisModuleOnly := FALSE);

	E_PMLUnitMode.ePMLUnitMode_Maintenance:
		AllowHMIControl(ThisModuleOnly := FALSE);
END_CASE
END_METHOD

METHOD PROTECTED HoldImmediate
VAR_INPUT
END_VAR
ChangeState(E_PMLCommand.ePMLCommand_Hold);
END_METHOD

METHOD PROTECTED Holding
VAR_INPUT
END_VAR
CASE _CurrentMode OF
	//=================================PRODUCTION MODE==================================
	E_PMLUnitMode.ePMLUnitMode_Production:
	//	IF (Sealer.CurrentState = E_PMLState.ePMLState_Complete OR Sealer.CurrentState = E_PMLState.ePMLState_Idle) AND (PullWheels.CurrentState = E_PMLState.ePMLState_Complete OR PullWheels.CurrentState = E_PMLState.ePMLState_Idle) THEN
			StateComplete();
	//	END_IF

	E_PMLUnitMode.ePMLUnitMode_Maintenance, E_PMLUnitMode.ePMLUnitMode_Manual:
		SUPER^.Holding();
END_CASE
END_METHOD

METHOD PROTECTED Initialize : BOOL
VAR
	i : UDINT; //Generic iteration value
END_VAR
Initialize := FALSE;
CASE DescendantSequenceState OF
	0:
	//	RegisterSubmodule(Safety_SubModule);		Disabled Needs IO issue resolving to allow estop circuit.
		RegisterSubmodule(Systems_SubModule);
	//	RegisterSubmodule(Closer_Gluer);
		RegisterSubmodule(Station_1);
		//RegisterSubmodule(Buffer_1);
//		RegisterSubmodule(Labeler);
	//	RegisterSubmodule(Diverter);
		RegisterSubmodule(Station_5);
		
		_LogModeChanges			:= FALSE;
		_LogStateChanges		:= FALSE;
		DescendantSequenceState := DescendantSequenceState + 10;

	10:
		//Setup Custom modes here

		(*CustomModes(eMode                          :=,
                    sName                          :=,
                    bDisableClearing               :=,
                    bDisableStarting               :=,
                    bDisableSuspended              :=,
                    bDisableStopping               :=,
                    bDisableAborting               :=,
                    bDisableHolding                :=,
                    bDisableHeld                   :=,
                    bDisableUnholding              :=,
                    bDisableSuspending             :=,
                    bDisableUnsuspending           :=,
                    bDisableResetting              :=,
                    bDisableIdle                   :=,
                    bDisableCompleting             :=,
                    bDisableComplete               :=,
                    bEnableUnitModeChangeStopped   :=,
                    bEnableUnitModeChangeIdle      :=,
                    bEnableUnitModeChangeSuspended :=,
                    bEnableUnitModeChangeExecute   :=,
                    bEnableUnitModeChangeAborted   :=,
                    bEnableUnitModeChangeHeld      :=,
                    bEnableUnitModeChangeComplete  :=,
                    bError                         =>,
                    nErrorId                       =>);*)
		DescendantSequenceState := DescendantSequenceState + 10;

	20:
		//Copy Mode names
		FOR i := 1 TO 3 DO
			ModeNames[i] := F_UnitModeToString(UDINT_TO_DINT(i));
		END_FOR

		DescendantSequenceState := DescendantSequenceState + 10;

	30:
		// Initialize Recipes 
		Initialize_Recipes();
		DescendantSequenceState := DescendantSequenceState + 10;

	40:
		//Call the Super
		IF SUPER^.Initialize() THEN
			DescendantSequenceState := DescendantSequenceState + 10;
		END_IF

	50:
		Initialize := TRUE;
END_CASE
END_METHOD

METHOD Initialize_Recipes
VAR_INPUT
END_VAR
// configuration of parameters Max Speed
_packTags.Command.Parameter[1].ID	 := 1;
_packTags.Command.Parameter[1].Name	 := 'Max Speed';
_packTags.Command.Parameter[1].Unit	 := '/min';
_packTags.Command.Parameter[1].Value := 180;
_packTags.Command.Parameter[2].ID	 := 2;
_packTags.Command.Parameter[2].Name	 := 'Product to Run';
_packTags.Command.Parameter[2].Unit	 := '';
_packTags.Command.Parameter[2].Value := 1;

// Recipe Product 1
_PackTags.Command.Product[1].ProductID								:= 100;
_PackTags.Command.Product[1].Ingredients[1].IngredientID			:= 1;
_PackTags.Command.Product[1].Ingredients[1].Parameter[1].ID			:= _PackTags.Command.Product[1].ProductID * 10 + 1;
_PackTags.Command.Product[1].Ingredients[1].Parameter[1].Name		:= 'Material Type';
_PackTags.Command.Product[1].Ingredients[1].Parameter[1].Unit		:= 'n/a';
_PackTags.Command.Product[1].Ingredients[1].Parameter[1].Value		:= 5;
_PackTags.Command.Product[1].Ingredients[1].Parameter[2].ID			:= _PackTags.Command.Product[1].ProductID * 10 + 2;
_PackTags.Command.Product[1].Ingredients[1].Parameter[2].Name		:= 'Material Thickness';
_PackTags.Command.Product[1].Ingredients[1].Parameter[2].Unit		:= 'um';
_PackTags.Command.Product[1].Ingredients[1].Parameter[2].Value		:= 240;
_PackTags.Command.Product[1].ProcessVariables[LENGTH].ID			:= _PackTags.Command.Product[1].ProductID * 20 + 1;
_PackTags.Command.Product[1].ProcessVariables[LENGTH].Name			:= 'Length';
_PackTags.Command.Product[1].ProcessVariables[LENGTH].Unit			:= 'mm';
_PackTags.Command.Product[1].ProcessVariables[LENGTH].Value			:= 100;
_PackTags.Command.Product[1].ProcessVariables[SEALTEMP].ID			:= _PackTags.Command.Product[1].ProductID * 20 + 2;
_PackTags.Command.Product[1].ProcessVariables[SEALTEMP].Name		:= 'Sealing Temp';
_PackTags.Command.Product[1].ProcessVariables[SEALTEMP].Unit		:= 'C';
_PackTags.Command.Product[1].ProcessVariables[SEALTEMP].Value		:= 100;
_PackTags.Command.Product[1].ProcessVariables[SEALTIME].ID			:= _PackTags.Command.Product[1].ProductID * 20 + 3;
_PackTags.Command.Product[1].ProcessVariables[SEALTIME].Name		:= 'Sealing Time';
_PackTags.Command.Product[1].ProcessVariables[SEALTIME].Unit		:= 'ms';
_PackTags.Command.Product[1].ProcessVariables[SEALTIME].Value		:= 50;
_PackTags.Command.Product[1].ProcessVariables[PULLWHEELS_VEL].ID	:= _PackTags.Command.Product[1].ProductID * 20 + 4;
_PackTags.Command.Product[1].ProcessVariables[PULLWHEELS_VEL].Name	:= 'Pull Wheels Vel';
_PackTags.Command.Product[1].ProcessVariables[PULLWHEELS_VEL].Unit	:= 'mm/s';
_PackTags.Command.Product[1].ProcessVariables[PULLWHEELS_VEL].Value := 100;
_PackTags.Command.Product[1].ProcessVariables[PULLWHEELS_ACC].ID	:= _PackTags.Command.Product[1].ProductID * 20 + 5;
_PackTags.Command.Product[1].ProcessVariables[PULLWHEELS_ACC].Name	:= 'Pull Wheels Acc';
_PackTags.Command.Product[1].ProcessVariables[PULLWHEELS_ACC].Unit	:= 'mm/s2';
_PackTags.Command.Product[1].ProcessVariables[PULLWHEELS_ACC].Value := 1000;
_PackTags.Command.Product[1].ProcessVariables[OPEN_POS].ID			:= _PackTags.Command.Product[1].ProductID * 20 + 6;
_PackTags.Command.Product[1].ProcessVariables[OPEN_POS].Name		:= 'Sealer Open Position';
_PackTags.Command.Product[1].ProcessVariables[OPEN_POS].Unit		:= 'mm';
_PackTags.Command.Product[1].ProcessVariables[OPEN_POS].Value		:= 105;
_PackTags.Command.Product[1].ProcessVariables[CLOSED_POS].ID		:= _PackTags.Command.Product[1].ProductID * 20 + 7;
_PackTags.Command.Product[1].ProcessVariables[CLOSED_POS].Name		:= 'Sealer Closed Position';
_PackTags.Command.Product[1].ProcessVariables[CLOSED_POS].Unit		:= 'mm';
_PackTags.Command.Product[1].ProcessVariables[CLOSED_POS].Value		:= 250;
_PackTags.Command.Product[1].ProcessVariables[SEALER_VEL].ID		:= _PackTags.Command.Product[1].ProductID * 20 + 8;
_PackTags.Command.Product[1].ProcessVariables[SEALER_VEL].Name		:= 'Sealer Vel';
_PackTags.Command.Product[1].ProcessVariables[SEALER_VEL].Unit		:= 'mm/s';
_PackTags.Command.Product[1].ProcessVariables[SEALER_VEL].Value		:= 100;
_PackTags.Command.Product[1].ProcessVariables[SEALER_ACC].ID		:= _PackTags.Command.Product[1].ProductID * 20 + 9;
_PackTags.Command.Product[1].ProcessVariables[SEALER_ACC].Name		:= 'Sealer Acc';
_PackTags.Command.Product[1].ProcessVariables[SEALER_ACC].Unit		:= 'mm/s2';
_PackTags.Command.Product[1].ProcessVariables[SEALER_ACC].Value		:= 1000;
_PackTags.Command.Product[1].ProcessVariables[UNWIND_VEL].ID		:= _PackTags.Command.Product[1].ProductID * 20 + 10;
_PackTags.Command.Product[1].ProcessVariables[UNWIND_VEL].Name		:= 'Unwind Vel';
_PackTags.Command.Product[1].ProcessVariables[UNWIND_VEL].Unit		:= 'mm/s';
_PackTags.Command.Product[1].ProcessVariables[UNWIND_VEL].Value		:= 100;
_PackTags.Command.Product[1].ProcessVariables[UNWIND_ACC].ID		:= _PackTags.Command.Product[1].ProductID * 20 + 11;
_PackTags.Command.Product[1].ProcessVariables[UNWIND_ACC].Name		:= 'Unwind Acc';
_PackTags.Command.Product[1].ProcessVariables[UNWIND_ACC].Unit		:= 'mm/s2';
_PackTags.Command.Product[1].ProcessVariables[UNWIND_ACC].Value		:= 1000;

// Product 2
_PackTags.Command.Product[2].ProductID								:= 100;
_PackTags.Command.Product[2].Ingredients[1].IngredientID			:= 1;
_PackTags.Command.Product[2].Ingredients[1].Parameter[1].ID			:= _PackTags.Command.Product[1].ProductID * 10 + 1;
_PackTags.Command.Product[2].Ingredients[1].Parameter[1].Name		:= 'Material Type';
_PackTags.Command.Product[2].Ingredients[1].Parameter[1].Unit		:= 'n/a';
_PackTags.Command.Product[2].Ingredients[1].Parameter[1].Value		:= 2;
_PackTags.Command.Product[2].Ingredients[1].Parameter[2].ID			:= _PackTags.Command.Product[1].ProductID * 10 + 2;
_PackTags.Command.Product[2].Ingredients[1].Parameter[2].Name		:= 'Material Thickness';
_PackTags.Command.Product[2].Ingredients[1].Parameter[2].Unit		:= 'um';
_PackTags.Command.Product[2].Ingredients[1].Parameter[2].Value		:= 220;
_PackTags.Command.Product[2].ProcessVariables[LENGTH].ID			:= _PackTags.Command.Product[1].ProductID * 20 + 1;
_PackTags.Command.Product[2].ProcessVariables[LENGTH].Name			:= 'Length';
_PackTags.Command.Product[2].ProcessVariables[LENGTH].Unit			:= 'mm';
_PackTags.Command.Product[2].ProcessVariables[LENGTH].Value			:= 55;
_PackTags.Command.Product[2].ProcessVariables[SEALTEMP].ID			:= _PackTags.Command.Product[1].ProductID * 20 + 2;
_PackTags.Command.Product[2].ProcessVariables[SEALTEMP].Name		:= 'Sealing Temp';
_PackTags.Command.Product[2].ProcessVariables[SEALTEMP].Unit		:= 'C';
_PackTags.Command.Product[2].ProcessVariables[SEALTEMP].Value		:= 110;
_PackTags.Command.Product[2].ProcessVariables[SEALTIME].ID			:= _PackTags.Command.Product[1].ProductID * 20 + 3;
_PackTags.Command.Product[2].ProcessVariables[SEALTIME].Name		:= 'Sealing Time';
_PackTags.Command.Product[2].ProcessVariables[SEALTIME].Unit		:= 'ms';
_PackTags.Command.Product[2].ProcessVariables[SEALTIME].Value		:= 100;
_PackTags.Command.Product[2].ProcessVariables[PULLWHEELS_VEL].ID	:= _PackTags.Command.Product[1].ProductID * 20 + 4;
_PackTags.Command.Product[2].ProcessVariables[PULLWHEELS_VEL].Name	:= 'Pull Wheels Vel';
_PackTags.Command.Product[2].ProcessVariables[PULLWHEELS_VEL].Unit	:= 'mm/s';
_PackTags.Command.Product[2].ProcessVariables[PULLWHEELS_VEL].Value := 200;
_PackTags.Command.Product[2].ProcessVariables[PULLWHEELS_ACC].ID	:= _PackTags.Command.Product[1].ProductID * 20 + 5;
_PackTags.Command.Product[2].ProcessVariables[PULLWHEELS_ACC].Name	:= 'Pull Wheels Acc';
_PackTags.Command.Product[2].ProcessVariables[PULLWHEELS_ACC].Unit	:= 'mm/s2';
_PackTags.Command.Product[2].ProcessVariables[PULLWHEELS_ACC].Value := 2000;
_PackTags.Command.Product[2].ProcessVariables[OPEN_POS].ID			:= _PackTags.Command.Product[1].ProductID * 20 + 6;
_PackTags.Command.Product[2].ProcessVariables[OPEN_POS].Name		:= 'Sealer Open Position';
_PackTags.Command.Product[2].ProcessVariables[OPEN_POS].Unit		:= 'mm';
_PackTags.Command.Product[2].ProcessVariables[OPEN_POS].Value		:= 60;
_PackTags.Command.Product[2].ProcessVariables[CLOSED_POS].ID		:= _PackTags.Command.Product[1].ProductID * 20 + 7;
_PackTags.Command.Product[2].ProcessVariables[CLOSED_POS].Name		:= 'Sealer Closed Position';
_PackTags.Command.Product[2].ProcessVariables[CLOSED_POS].Unit		:= 'mm';
_PackTags.Command.Product[2].ProcessVariables[CLOSED_POS].Value		:= 253;
_PackTags.Command.Product[2].ProcessVariables[SEALER_VEL].ID		:= _PackTags.Command.Product[1].ProductID * 20 + 8;
_PackTags.Command.Product[2].ProcessVariables[SEALER_VEL].Name		:= 'Sealer Vel';
_PackTags.Command.Product[2].ProcessVariables[SEALER_VEL].Unit		:= 'mm/s';
_PackTags.Command.Product[2].ProcessVariables[SEALER_VEL].Value		:= 200;
_PackTags.Command.Product[2].ProcessVariables[SEALER_ACC].ID		:= _PackTags.Command.Product[1].ProductID * 20 + 9;
_PackTags.Command.Product[2].ProcessVariables[SEALER_ACC].Name		:= 'Sealer Acc';
_PackTags.Command.Product[2].ProcessVariables[SEALER_ACC].Unit		:= 'mm/s2';
_PackTags.Command.Product[2].ProcessVariables[SEALER_ACC].Value		:= 2000;
_PackTags.Command.Product[2].ProcessVariables[UNWIND_VEL].ID		:= _PackTags.Command.Product[1].ProductID * 20 + 10;
_PackTags.Command.Product[2].ProcessVariables[UNWIND_VEL].Name		:= 'Unwind Vel';
_PackTags.Command.Product[2].ProcessVariables[UNWIND_VEL].Unit		:= 'mm/s';
_PackTags.Command.Product[2].ProcessVariables[UNWIND_VEL].Value		:= 200;
_PackTags.Command.Product[2].ProcessVariables[UNWIND_ACC].ID		:= _PackTags.Command.Product[1].ProductID * 20 + 11;
_PackTags.Command.Product[2].ProcessVariables[UNWIND_ACC].Name		:= 'Unwind Acc';
_PackTags.Command.Product[2].ProcessVariables[UNWIND_ACC].Unit		:= 'mm/s2';
_PackTags.Command.Product[2].ProcessVariables[UNWIND_ACC].Value		:= 2000;

//Product 3
_PackTags.Command.Product[3].ProductID								:= 307;
_PackTags.Command.Product[3].Ingredients[1].IngredientID			:= 1;
_PackTags.Command.Product[3].Ingredients[1].Parameter[1].ID			:= _PackTags.Command.Product[1].ProductID * 10 + 1;
_PackTags.Command.Product[3].Ingredients[1].Parameter[1].Name		:= 'Material Type';
_PackTags.Command.Product[3].Ingredients[1].Parameter[1].Unit		:= 'n/a';
_PackTags.Command.Product[3].Ingredients[1].Parameter[1].Value		:= 2;
_PackTags.Command.Product[3].Ingredients[1].Parameter[2].ID			:= _PackTags.Command.Product[1].ProductID * 10 + 2;
_PackTags.Command.Product[3].Ingredients[1].Parameter[2].Name		:= 'Material Thickness';
_PackTags.Command.Product[3].Ingredients[1].Parameter[2].Unit		:= 'um';
_PackTags.Command.Product[3].Ingredients[1].Parameter[2].Value		:= 220;
_PackTags.Command.Product[3].ProcessVariables[LENGTH].ID			:= _PackTags.Command.Product[1].ProductID * 20 + 1;
_PackTags.Command.Product[3].ProcessVariables[LENGTH].Name			:= 'Length';
_PackTags.Command.Product[3].ProcessVariables[LENGTH].Unit			:= 'mm';
_PackTags.Command.Product[3].ProcessVariables[LENGTH].Value			:= 85;
_PackTags.Command.Product[3].ProcessVariables[SEALTEMP].ID			:= _PackTags.Command.Product[1].ProductID * 20 + 2;
_PackTags.Command.Product[3].ProcessVariables[SEALTEMP].Name		:= 'Sealing Temp';
_PackTags.Command.Product[3].ProcessVariables[SEALTEMP].Unit		:= 'C';
_PackTags.Command.Product[3].ProcessVariables[SEALTEMP].Value		:= 95;
_PackTags.Command.Product[3].ProcessVariables[SEALTIME].ID			:= _PackTags.Command.Product[1].ProductID * 20 + 3;
_PackTags.Command.Product[3].ProcessVariables[SEALTIME].Name		:= 'Sealing Time';
_PackTags.Command.Product[3].ProcessVariables[SEALTIME].Unit		:= 'ms';
_PackTags.Command.Product[3].ProcessVariables[SEALTIME].Value		:= 20;
_PackTags.Command.Product[3].ProcessVariables[PULLWHEELS_VEL].ID	:= _PackTags.Command.Product[1].ProductID * 20 + 4;
_PackTags.Command.Product[3].ProcessVariables[PULLWHEELS_VEL].Name	:= 'Pull Wheels Vel';
_PackTags.Command.Product[3].ProcessVariables[PULLWHEELS_VEL].Unit	:= 'mm/s';
_PackTags.Command.Product[3].ProcessVariables[PULLWHEELS_VEL].Value := 300;
_PackTags.Command.Product[3].ProcessVariables[PULLWHEELS_ACC].ID	:= _PackTags.Command.Product[1].ProductID * 20 + 5;
_PackTags.Command.Product[3].ProcessVariables[PULLWHEELS_ACC].Name	:= 'Pull Wheels Acc';
_PackTags.Command.Product[3].ProcessVariables[PULLWHEELS_ACC].Unit	:= 'mm/s2';
_PackTags.Command.Product[3].ProcessVariables[PULLWHEELS_ACC].Value := 3000;
_PackTags.Command.Product[3].ProcessVariables[OPEN_POS].ID			:= _PackTags.Command.Product[1].ProductID * 20 + 6;
_PackTags.Command.Product[3].ProcessVariables[OPEN_POS].Name		:= 'Sealer Open Position';
_PackTags.Command.Product[3].ProcessVariables[OPEN_POS].Unit		:= 'mm';
_PackTags.Command.Product[3].ProcessVariables[OPEN_POS].Value		:= 56;
_PackTags.Command.Product[3].ProcessVariables[CLOSED_POS].ID		:= _PackTags.Command.Product[1].ProductID * 20 + 7;
_PackTags.Command.Product[3].ProcessVariables[CLOSED_POS].Name		:= 'Sealer Closed Position';
_PackTags.Command.Product[3].ProcessVariables[CLOSED_POS].Unit		:= 'mm';
_PackTags.Command.Product[3].ProcessVariables[CLOSED_POS].Value		:= 265;
_PackTags.Command.Product[3].ProcessVariables[SEALER_VEL].ID		:= _PackTags.Command.Product[1].ProductID * 20 + 8;
_PackTags.Command.Product[3].ProcessVariables[SEALER_VEL].Name		:= 'Sealer Vel';
_PackTags.Command.Product[3].ProcessVariables[SEALER_VEL].Unit		:= 'mm/s';
_PackTags.Command.Product[3].ProcessVariables[SEALER_VEL].Value		:= 300;
_PackTags.Command.Product[3].ProcessVariables[SEALER_ACC].ID		:= _PackTags.Command.Product[1].ProductID * 20 + 9;
_PackTags.Command.Product[3].ProcessVariables[SEALER_ACC].Name		:= 'Sealer Acc';
_PackTags.Command.Product[3].ProcessVariables[SEALER_ACC].Unit		:= 'mm/s2';
_PackTags.Command.Product[3].ProcessVariables[SEALER_ACC].Value		:= 3000;
_PackTags.Command.Product[3].ProcessVariables[UNWIND_VEL].ID		:= _PackTags.Command.Product[1].ProductID * 20 + 10;
_PackTags.Command.Product[3].ProcessVariables[UNWIND_VEL].Name		:= 'Unwind Vel';
_PackTags.Command.Product[3].ProcessVariables[UNWIND_VEL].Unit		:= 'mm/s';
_PackTags.Command.Product[3].ProcessVariables[UNWIND_VEL].Value		:= 300;
_PackTags.Command.Product[3].ProcessVariables[UNWIND_ACC].ID		:= _PackTags.Command.Product[1].ProductID * 20 + 11;
_PackTags.Command.Product[3].ProcessVariables[UNWIND_ACC].Name		:= 'Unwind Acc';
_PackTags.Command.Product[3].ProcessVariables[UNWIND_ACC].Unit		:= 'mm/s2';
_PackTags.Command.Product[3].ProcessVariables[UNWIND_ACC].Value		:= 3000;

//Product 4
_PackTags.Command.Product[4].ProductID								:= 401;
_PackTags.Command.Product[4].Ingredients[1].IngredientID			:= 1;
_PackTags.Command.Product[4].Ingredients[1].Parameter[1].ID			:= _PackTags.Command.Product[1].ProductID * 10 + 1;
_PackTags.Command.Product[4].Ingredients[1].Parameter[1].Name		:= 'Material Type';
_PackTags.Command.Product[4].Ingredients[1].Parameter[1].Unit		:= 'n/a';
_PackTags.Command.Product[4].Ingredients[1].Parameter[1].Value		:= 2;
_PackTags.Command.Product[4].Ingredients[1].Parameter[2].ID			:= _PackTags.Command.Product[1].ProductID * 10 + 2;
_PackTags.Command.Product[4].Ingredients[1].Parameter[2].Name		:= 'Material Thickness';
_PackTags.Command.Product[4].Ingredients[1].Parameter[2].Unit		:= 'um';
_PackTags.Command.Product[4].Ingredients[1].Parameter[2].Value		:= 220;
_PackTags.Command.Product[4].ProcessVariables[LENGTH].ID			:= _PackTags.Command.Product[1].ProductID * 20 + 1;
_PackTags.Command.Product[4].ProcessVariables[LENGTH].Name			:= 'Length';
_PackTags.Command.Product[4].ProcessVariables[LENGTH].Unit			:= 'mm';
_PackTags.Command.Product[4].ProcessVariables[LENGTH].Value			:= 85;
_PackTags.Command.Product[4].ProcessVariables[SEALTEMP].ID			:= _PackTags.Command.Product[1].ProductID * 20 + 2;
_PackTags.Command.Product[4].ProcessVariables[SEALTEMP].Name		:= 'Sealing Temp';
_PackTags.Command.Product[4].ProcessVariables[SEALTEMP].Unit		:= 'C';
_PackTags.Command.Product[4].ProcessVariables[SEALTEMP].Value		:= 95;
_PackTags.Command.Product[4].ProcessVariables[SEALTIME].ID			:= _PackTags.Command.Product[1].ProductID * 20 + 3;
_PackTags.Command.Product[4].ProcessVariables[SEALTIME].Name		:= 'Sealing Time';
_PackTags.Command.Product[4].ProcessVariables[SEALTIME].Unit		:= 'ms';
_PackTags.Command.Product[4].ProcessVariables[SEALTIME].Value		:= 80;
_PackTags.Command.Product[4].ProcessVariables[PULLWHEELS_VEL].ID	:= _PackTags.Command.Product[1].ProductID * 20 + 4;
_PackTags.Command.Product[4].ProcessVariables[PULLWHEELS_VEL].Name	:= 'Pull Wheels Vel';
_PackTags.Command.Product[4].ProcessVariables[PULLWHEELS_VEL].Unit	:= 'mm/s';
_PackTags.Command.Product[4].ProcessVariables[PULLWHEELS_VEL].Value := 100;
_PackTags.Command.Product[4].ProcessVariables[PULLWHEELS_ACC].ID	:= _PackTags.Command.Product[1].ProductID * 20 + 5;
_PackTags.Command.Product[4].ProcessVariables[PULLWHEELS_ACC].Name	:= 'Pull Wheels Acc';
_PackTags.Command.Product[4].ProcessVariables[PULLWHEELS_ACC].Unit	:= 'mm/s2';
_PackTags.Command.Product[4].ProcessVariables[PULLWHEELS_ACC].Value := 1000;
_PackTags.Command.Product[4].ProcessVariables[OPEN_POS].ID			:= _PackTags.Command.Product[1].ProductID * 20 + 6;
_PackTags.Command.Product[4].ProcessVariables[OPEN_POS].Name		:= 'Sealer Open Position';
_PackTags.Command.Product[4].ProcessVariables[OPEN_POS].Unit		:= 'mm';
_PackTags.Command.Product[4].ProcessVariables[OPEN_POS].Value		:= 105;
_PackTags.Command.Product[4].ProcessVariables[CLOSED_POS].ID		:= _PackTags.Command.Product[1].ProductID * 20 + 7;
_PackTags.Command.Product[4].ProcessVariables[CLOSED_POS].Name		:= 'Sealer Closed Position';
_PackTags.Command.Product[4].ProcessVariables[CLOSED_POS].Unit		:= 'mm';
_PackTags.Command.Product[4].ProcessVariables[CLOSED_POS].Value		:= 250;
_PackTags.Command.Product[4].ProcessVariables[SEALER_VEL].ID		:= _PackTags.Command.Product[1].ProductID * 20 + 8;
_PackTags.Command.Product[4].ProcessVariables[SEALER_VEL].Name		:= 'Sealer Vel';
_PackTags.Command.Product[4].ProcessVariables[SEALER_VEL].Unit		:= 'mm/s';
_PackTags.Command.Product[4].ProcessVariables[SEALER_VEL].Value		:= 100;
_PackTags.Command.Product[4].ProcessVariables[SEALER_ACC].ID		:= _PackTags.Command.Product[1].ProductID * 20 + 9;
_PackTags.Command.Product[4].ProcessVariables[SEALER_ACC].Name		:= 'Sealer Acc';
_PackTags.Command.Product[4].ProcessVariables[SEALER_ACC].Unit		:= 'mm/s2';
_PackTags.Command.Product[4].ProcessVariables[SEALER_ACC].Value		:= 1000;
_PackTags.Command.Product[4].ProcessVariables[UNWIND_VEL].ID		:= _PackTags.Command.Product[1].ProductID * 20 + 10;
_PackTags.Command.Product[4].ProcessVariables[UNWIND_VEL].Name		:= 'Unwind Vel';
_PackTags.Command.Product[4].ProcessVariables[UNWIND_VEL].Unit		:= 'mm/s';
_PackTags.Command.Product[4].ProcessVariables[UNWIND_VEL].Value		:= 100;
_PackTags.Command.Product[4].ProcessVariables[UNWIND_ACC].ID		:= _PackTags.Command.Product[1].ProductID * 20 + 11;
_PackTags.Command.Product[4].ProcessVariables[UNWIND_ACC].Name		:= 'Unwind Acc';
_PackTags.Command.Product[4].ProcessVariables[UNWIND_ACC].Unit		:= 'mm/s2';
_PackTags.Command.Product[4].ProcessVariables[UNWIND_ACC].Value		:= 1000;

//Product 5
_PackTags.Command.Product[5].ProductID								:= 522;
_PackTags.Command.Product[5].Ingredients[1].IngredientID			:= 1;
_PackTags.Command.Product[5].Ingredients[1].Parameter[1].ID			:= _PackTags.Command.Product[1].ProductID * 10 + 1;
_PackTags.Command.Product[5].Ingredients[1].Parameter[1].Name		:= 'Material Type';
_PackTags.Command.Product[5].Ingredients[1].Parameter[1].Unit		:= 'n/a';
_PackTags.Command.Product[5].Ingredients[1].Parameter[1].Value		:= 2;
_PackTags.Command.Product[5].Ingredients[1].Parameter[2].ID			:= _PackTags.Command.Product[1].ProductID * 10 + 2;
_PackTags.Command.Product[5].Ingredients[1].Parameter[2].Name		:= 'Material Thickness';
_PackTags.Command.Product[5].Ingredients[1].Parameter[2].Unit		:= 'um';
_PackTags.Command.Product[5].Ingredients[1].Parameter[2].Value		:= 520;
_PackTags.Command.Product[5].ProcessVariables[LENGTH].ID			:= _PackTags.Command.Product[1].ProductID * 20 + 1;
_PackTags.Command.Product[5].ProcessVariables[LENGTH].Name			:= 'Length';
_PackTags.Command.Product[5].ProcessVariables[LENGTH].Unit			:= 'mm';
_PackTags.Command.Product[5].ProcessVariables[LENGTH].Value			:= 200;
_PackTags.Command.Product[5].ProcessVariables[SEALTEMP].ID			:= _PackTags.Command.Product[1].ProductID * 20 + 2;
_PackTags.Command.Product[5].ProcessVariables[SEALTEMP].Name		:= 'Sealing Temp';
_PackTags.Command.Product[5].ProcessVariables[SEALTEMP].Unit		:= 'C';
_PackTags.Command.Product[5].ProcessVariables[SEALTEMP].Value		:= 130;
_PackTags.Command.Product[5].ProcessVariables[SEALTIME].ID			:= _PackTags.Command.Product[1].ProductID * 20 + 3;
_PackTags.Command.Product[5].ProcessVariables[SEALTIME].Name		:= 'Sealing Time';
_PackTags.Command.Product[5].ProcessVariables[SEALTIME].Unit		:= 'ms';
_PackTags.Command.Product[5].ProcessVariables[SEALTIME].Value		:= 200;
_PackTags.Command.Product[5].ProcessVariables[PULLWHEELS_VEL].ID	:= _PackTags.Command.Product[1].ProductID * 20 + 4;
_PackTags.Command.Product[5].ProcessVariables[PULLWHEELS_VEL].Name	:= 'Pull Wheels Vel';
_PackTags.Command.Product[5].ProcessVariables[PULLWHEELS_VEL].Unit	:= 'mm/s';
_PackTags.Command.Product[5].ProcessVariables[PULLWHEELS_VEL].Value := 100;
_PackTags.Command.Product[5].ProcessVariables[PULLWHEELS_ACC].ID	:= _PackTags.Command.Product[1].ProductID * 20 + 5;
_PackTags.Command.Product[5].ProcessVariables[PULLWHEELS_ACC].Name	:= 'Pull Wheels Acc';
_PackTags.Command.Product[5].ProcessVariables[PULLWHEELS_ACC].Unit	:= 'mm/s2';
_PackTags.Command.Product[5].ProcessVariables[PULLWHEELS_ACC].Value := 1000;
_PackTags.Command.Product[5].ProcessVariables[OPEN_POS].ID			:= _PackTags.Command.Product[1].ProductID * 20 + 6;
_PackTags.Command.Product[5].ProcessVariables[OPEN_POS].Name		:= 'Sealer Open Position';
_PackTags.Command.Product[5].ProcessVariables[OPEN_POS].Unit		:= 'mm';
_PackTags.Command.Product[5].ProcessVariables[OPEN_POS].Value		:= 105;
_PackTags.Command.Product[5].ProcessVariables[CLOSED_POS].ID		:= _PackTags.Command.Product[1].ProductID * 20 + 7;
_PackTags.Command.Product[5].ProcessVariables[CLOSED_POS].Name		:= 'Sealer Closed Position';
_PackTags.Command.Product[5].ProcessVariables[CLOSED_POS].Unit		:= 'mm';
_PackTags.Command.Product[5].ProcessVariables[CLOSED_POS].Value		:= 250;
_PackTags.Command.Product[5].ProcessVariables[SEALER_VEL].ID		:= _PackTags.Command.Product[1].ProductID * 20 + 8;
_PackTags.Command.Product[5].ProcessVariables[SEALER_VEL].Name		:= 'Sealer Vel';
_PackTags.Command.Product[5].ProcessVariables[SEALER_VEL].Unit		:= 'mm/s';
_PackTags.Command.Product[5].ProcessVariables[SEALER_VEL].Value		:= 100;
_PackTags.Command.Product[5].ProcessVariables[SEALER_ACC].ID		:= _PackTags.Command.Product[1].ProductID * 20 + 9;
_PackTags.Command.Product[5].ProcessVariables[SEALER_ACC].Name		:= 'Sealer Acc';
_PackTags.Command.Product[5].ProcessVariables[SEALER_ACC].Unit		:= 'mm/s2';
_PackTags.Command.Product[5].ProcessVariables[SEALER_ACC].Value		:= 1000;
_PackTags.Command.Product[5].ProcessVariables[UNWIND_VEL].ID		:= _PackTags.Command.Product[1].ProductID * 20 + 10;
_PackTags.Command.Product[5].ProcessVariables[UNWIND_VEL].Name		:= 'Unwind Vel';
_PackTags.Command.Product[5].ProcessVariables[UNWIND_VEL].Unit		:= 'mm/s';
_PackTags.Command.Product[5].ProcessVariables[UNWIND_VEL].Value		:= 100;
_PackTags.Command.Product[5].ProcessVariables[UNWIND_ACC].ID		:= _PackTags.Command.Product[1].ProductID * 20 + 11;
_PackTags.Command.Product[5].ProcessVariables[UNWIND_ACC].Name		:= 'Unwind Acc';
_PackTags.Command.Product[5].ProcessVariables[UNWIND_ACC].Unit		:= 'mm/s2';
_PackTags.Command.Product[5].ProcessVariables[UNWIND_ACC].Value		:= 1000;
CurrentRecipeName													:= 'From PackTags';
END_METHOD

PROPERTY PUBLIC PackTags : ST_PackMLv30Ext
GET
PackTags := _packTags;
END_GET
END_PROPERTY

METHOD RaiseAlarm2Args
VAR_IN_OUT
	Alarm : FB_TcAlarm; //Alarm to be raised
END_VAR

VAR_INPUT
	String_1 : STRING; //First String Parameter (The Name of this component will be applied first automatically)
	String_2 : STRING; //Second String Parameter
END_VAR
F_RaiseAlarmWithStringParameters(Alarm	  := Alarm,
								 String_1 := Name,
								 String_2 := String_1,
								 String_3 := String_2);
END_METHOD

METHOD PROTECTED Resetting
VAR_INPUT
END_VAR
CASE _CurrentMode OF
	//=================================PRODUCTION MODE==================================
	E_PMLUnitMode.ePMLUnitMode_Production:
		IF DataFromPackML THEN
			product					:= LREAL_TO_INT(_PackTags.Command.Parameter[2].Value);
	//		Buffer_1.Velocity		:= LREAL_TO_INT(_PackTags.Command.Product[product].ProcessVariables[PULLWHEELS_VEL].Value);
//			PullWheels.Length		:= _PackTags.Command.Product[product].ProcessVariables[LENGTH].Value;
//			PullWheels.Velocity		:= _PackTags.Command.Product[product].ProcessVariables[PULLWHEELS_VEL].Value;
//			PullWheels.Acceleration := _PackTags.Command.Product[product].ProcessVariables[PULLWHEELS_ACC].Value;
//			Sealer.SealTime			:= _PackTags.Command.Product[product].ProcessVariables[SEALTIME].Value;
//			Sealer.Temp				:= _PackTags.Command.Product[product].ProcessVariables[SEALTEMP].Value;
//			Sealer.OpenPos			:= _PackTags.Command.Product[product].ProcessVariables[OPEN_POS].Value;
//			Sealer.ClosedPos		:= _PackTags.Command.Product[product].ProcessVariables[CLOSED_POS].Value;
//			Sealer.Velocity			:= _PackTags.Command.Product[product].ProcessVariables[SEALER_VEL].Value;
//			Sealer.Acceleration		:= _PackTags.Command.Product[product].ProcessVariables[SEALER_ACC].Value;
//			Unwind.Velocity			:= _PackTags.Command.Product[product].ProcessVariables[UNWIND_VEL].Value;
//			Unwind.Acceleration		:= _PackTags.Command.Product[product].ProcessVariables[UNWIND_ACC].Value;
		END_IF

	E_PMLUnitMode.ePMLUnitMode_Maintenance, E_PMLUnitMode.ePMLUnitMode_Manual:
		;
END_CASE

SUPER^.Resetting();
END_METHOD

METHOD PROTECTED Starting
VAR_INPUT
END_VAR
CASE _CurrentMode OF
	//=================================PRODUCTION MODE==================================
	E_PMLUnitMode.ePMLUnitMode_Production:
		// The seal bar can go to Execute, the others will be run in Mahcine Execute
	//	Sealer.Heat := TRUE;
		StateComplete();

	E_PMLUnitMode.ePMLUnitMode_Maintenance, E_PMLUnitMode.ePMLUnitMode_Manual:
		SUPER^.Starting();
END_CASE
END_METHOD

METHOD PROTECTED Stopping
VAR_INPUT
END_VAR
CASE _CurrentMode OF
    //=================================PRODUCTION MODE==================================
    E_PMLUnitMode.ePMLUnitMode_Production:
        CASE SequenceState OF
            0:
                NoStateTasksToComplete := FALSE;
        		Station_1.ChangeState(E_PMLCommand.ePMLCommand_Stop);
                SequenceState := SequenceState + 10;
            10:
               IF Station_1.CurrentState = E_PMLState.ePMLState_Stopped THEN
		//		   Brakes.ChangeState(E_PMLCommand.ePMLCommand_Stop);
                    SequenceState := SequenceState + 10;
               END_IF
            20:
		//		IF Brakes.CurrentState = E_PMLState.ePMLState_Stopped THEN
						ChangeState(E_PMLCommand.ePMLCommand_Stop);
						StateTasksComplete := TRUE;
		//		END_IF
	  
        END_CASE

    //=================================MAINTENANCE & MANUAL MODE==================================
    E_PMLUnitMode.ePMLUnitMode_Maintenance, E_PMLUnitMode.ePMLUnitMode_Manual:
        ;
END_CASE

SUPER^.Stopping();


(*
20:	//Controlled shut down Contactoe then Brakes
					Generation.ChangeState(E_PMLCommand.ePMLCommand_Stop);
					SequenceState := SequenceState + 10;	
				30:
					IF Generation.CurrentState = E_PMLState.ePMLState_Stopped THEN
						Brakes.ChangeState(E_PMLCommand.ePMLCommand_Stop);
						SequenceState := SequenceState + 10;	
					END_IF
				40:
					IF Brakes.CurrentState = E_PMLState.ePMLState_Stopped THEN
						ChangeState(E_PMLCommand.ePMLCommand_Stop);
					END_IF*)
END_METHOD

METHOD PROTECTED SubModuleMonitor : BOOL
VAR
	AlarmResponses : ARRAY[0..4] OF E_AlarmResponse; //Temporary response array	
END_VAR
// Check the sub Modules for Alarm Severity
SUPER^.SubModuleMonitor();

//Check the alarms at the machine level
_CurrentAlarmSeverity := F_GetMaxSeverityRaised(Alarms := MachineAlarms, CurrentSeverity := _CurrentAlarmSeverity);

//Check the severity of the machine level alarms
IF _CurrentState <> E_PMLState.ePMLState_Aborted AND _CurrentState <> E_PMLState.ePMLState_Aborting AND _CurrentState <> E_PMLState.ePMLState_Clearing AND _CurrentState <> E_PMLState.ePMLState_Stopped AND _CurrentState <> E_PMLState.ePMLState_Stopping THEN
	AlarmResponses := _ParentFaultResponseDefinitions;
	CASE AlarmResponses[CurrentAlarmSeverity] OF
		E_AlarmResponse.Abort_ImmediateError:
			AbortImmediateError(Name, TRUE);

		E_AlarmResponse.Abort_Immediate:
			AbortImmediate();

		E_AlarmResponse.Stop_Immediate:
			StopImmediate();

		E_AlarmResponse.Stop_Controlled:
			StopControlled();

		E_AlarmResponse.Hold_Immediate:
			HoldImmediate();

		E_AlarmResponse.Suspend_Immediate:
			SuspendImmediate();

		E_AlarmResponse.Suspend_Controlled:
			SuspendControlled();

		E_AlarmResponse.NoResponse:
			;
	END_CASE
ELSIF _CurrentState = E_PMLState.ePMLState_Stopped OR _CurrentState = E_PMLState.ePMLState_Stopping THEN
	AlarmResponses := _ParentFaultResponseDefinitions;
	CASE AlarmResponses[CurrentAlarmSeverity] OF
		E_AlarmResponse.Abort_ImmediateError:
			AbortImmediateError(Name, TRUE);

		E_AlarmResponse.Abort_Immediate:
			AbortImmediate();

		E_AlarmResponse.NoResponse:
			;
	END_CASE
END_IF
END_METHOD

METHOD PROTECTED Suspended
VAR_INPUT
END_VAR
//IF THIS^.Sealer.sealbar.InTempRange THEN
	ChangeState(E_PMLCommand.ePMLCommand_Unsuspend);
//END_IF
END_METHOD

METHOD PROTECTED Suspending
VAR_INPUT
END_VAR
CASE _CurrentMode OF
	//=================================PRODUCTION MODE==================================
	E_PMLUnitMode.ePMLUnitMode_Production:
	//	IF (Sealer.CurrentState = E_PMLState.ePMLState_Complete OR Sealer.CurrentState = E_PMLState.ePMLState_Idle) AND (PullWheels.CurrentState = E_PMLState.ePMLState_Complete OR PullWheels.CurrentState = E_PMLState.ePMLState_Idle) THEN
			StateComplete();
	//	END_IF

	E_PMLUnitMode.ePMLUnitMode_Maintenance, E_PMLUnitMode.ePMLUnitMode_Manual:
		SUPER^.Suspending();
END_CASE
END_METHOD

METHOD PROTECTED Unholding
VAR_INPUT
END_VAR
CASE _CurrentMode OF
	//=================================PRODUCTION MODE==================================
	E_PMLUnitMode.ePMLUnitMode_Production:
		StateComplete();

	E_PMLUnitMode.ePMLUnitMode_Maintenance, E_PMLUnitMode.ePMLUnitMode_Manual:
		SUPER^.Unholding();
END_CASE
END_METHOD

METHOD PROTECTED Unsuspending
VAR_INPUT
END_VAR
CASE _CurrentMode OF
	//=================================PRODUCTION MODE==================================
	E_PMLUnitMode.ePMLUnitMode_Production:
		StateComplete();

	E_PMLUnitMode.ePMLUnitMode_Maintenance, E_PMLUnitMode.ePMLUnitMode_Manual:
		SUPER^.Unsuspending();
END_CASE
END_METHOD

METHOD UpdateModeTimers
VAR
	currentTime	 : T_DCTIME64;
	timeToUpdate : LREAL;
END_VAR

VAR_INST
	lastTime  : T_DCTIME64 := F_GetActualDcTime64();
	lastState : DINT;
	lastMode  : DINT;
END_VAR
IF _PackTags.Status.StateCurrent <> lastState THEN
	MEMSET(ADR(_PackTags.Admin.StateCurrentTime), 0, SIZEOF(_PackTags.Admin.StateCurrentTime));
	lastState := _PackTags.Status.StateCurrent;
END_IF

IF _PackTags.Status.UnitModeCurrent <> lastMode THEN
	MEMSET(ADR(_PackTags.Admin.ModeCurrentTime), 0, SIZEOF(_PackTags.Admin.ModeCurrentTime));
	lastMode := _PackTags.Status.UnitModeCurrent;
END_IF

currentTime := F_GetActualDcTime64();
IF lastTime <> 0 THEN
	timeToUpdate := ULINT_TO_LREAL(currentTime - lastTime) / 1_000_000_000.0;
END_IF

// only seconds get added to the cumulative timers 
IF timeToUpdate > 1 THEN
	_PackTags.Admin.ModeCummulativeTime[_PackTags.Status.UnitModeCurrent]								  := _PackTags.Admin.ModeCummulativeTime[_PackTags.Status.UnitModeCurrent] + LREAL_TO_DINT(timeToUpdate);
	_PackTags.Admin.ModeCurrentTime[_PackTags.Status.UnitModeCurrent]									  := _PackTags.Admin.ModeCurrentTime[_PackTags.Status.UnitModeCurrent] + LREAL_TO_DINT(timeToUpdate);
	_PackTags.Admin.StateCummulativeTime[_PackTags.Status.UnitModeCurrent, _PackTags.Status.StateCurrent] := _PackTags.Admin.StateCummulativeTime[_PackTags.Status.UnitModeCurrent, _PackTags.Status.StateCurrent] + LREAL_TO_DINT(timeToUpdate);
	_PackTags.Admin.StateCurrentTime[_PackTags.Status.UnitModeCurrent, _PackTags.Status.StateCurrent]	  := _PackTags.Admin.StateCurrentTime[_PackTags.Status.UnitModeCurrent, _PackTags.Status.StateCurrent] + LREAL_TO_DINT(timeToUpdate);
	lastTime																							  := currentTime;
END_IF
END_METHOD

END_FUNCTION_BLOCK

// ---- Machine/SafetyModules/FB_Safety_Module.TcPOU
FUNCTION_BLOCK FB_Safety_Module EXTENDS FB_PackML_BaseModule // IMPLEMENTS I_ControlsProductionRate
VAR
	// Sub Modules
	
	// Components
	Reset_PB : FB_DigitalSensor		:= (Name := 'Reset PB', DebounceMode := E_DebounceMode.SimpleFlickerFilter, DebounceTime := T#250MS, Inverted    := FALSE, SimulationInput:= FALSE, SimulationMode := E_SensorSimulationMode.InputDriven) ;
	Safty_Reset_Pulse_Out : Relay(Invert_Output	:=FALSE);

	SafetyGroupAutoReset : FB_SafetyResetPulse;
	
	SafetyGroup_IO     : FB_Component_Safety_Group :=(
		Name := 'IO Group',
		SafetyReset := SafetyGroupAutoReset,
		AutoResetConnectionFaults := TRUE);
	
	SafetyGroup_ESTOP     : FB_Component_Safety_Group :=(
		Name := 'ESTOP Group',
		SafetyReset := SafetyGroupAutoReset,
		AutoResetConnectionFaults := TRUE);
	
	SafetyReset   : FB_SafetyResetPulse;
	SafetyOutput  : FB_Component_Safety_ConnectionFB :=(
		Name := 'Output Card 1 EL2904',
		DependenceFB := SafetyGroup_ESTOP,
		SafetyReset := SafetyReset);
		
	SafetyInput  : FB_Component_Safety_ConnectionFB :=(
		Name := 'Input Card 1 EL1904',
		DependenceFB := SafetyGroup_ESTOP,
		SafetyReset := SafetyReset);
////An instance of FB_Component_Safety_EstopFB can be declared as follows:


	SafetyEstop  : FB_Component_Safety_EstopFB  :=(
		Name := 'E-Stop',
		DependenceFB := SafetyOutput,
		SafetyReset := SafetyReset);	


	//Initial List of Components
	ipComponents_Init : ARRAY[1..Parameters_PackML_Base.MAX_NO_OF_COMPONENTS] OF I_ComponentBase := [];

	//Alarms for this module
	MachineSafetyAlarms : ARRAY[1..SAFETY_ALARM_COUNT] OF FB_TcAlarm;

	//Current Recipe Name
	CurrentRecipeName : STRING;

	//Get Data From PackML? Else RecipeManager is running
	DataFromPackML : BOOL := TRUE;

	//Data 
//	sealTimeStart : ULINT;
//	sealTimeEnd	  : ULINT;
//	sealingTime	  : LREAL;
//	sealTrig	  : R_TRIG;
//	pullTimeStart : ULINT;
//	pullTimeEnd	  : ULINT;
//	pullingTime	  : LREAL;
//	pulltrig	  : R_TRIG;
//	partTimeStart : ULINT;
//	partTimeEnd	  : ULINT;
//	partTime	  : LREAL;
//	parts		  : DINT;
//	product		  : DINT;

	//Pack Tags for System
	{attribute 'OPC.UA.DA' := '1'}
	_PackTags : ST_PackMLv30Ext; //ST_PackMLv30 is obsolete in Tc3_PackML_V2
END_VAR

VAR CONSTANT
	//PackTag parameter IDs
	LENGTH		   : INT := 1;
	SEALTEMP	   : INT := 2;
	SEALTIME	   : INT := 3;
	PULLWHEELS_VEL : INT := 4;
	PULLWHEELS_ACC : INT := 5;
	SEALER_VEL	   : INT := 6;
	SEALER_ACC	   : INT := 7;
	UNWIND_VEL	   : INT := 8;
	UNWIND_ACC	   : INT := 9;
	OPEN_POS	   : INT := 10;
	CLOSED_POS	   : INT := 11;

	//Alarm count constant
	SAFETY_ALARM_COUNT : INT := 6;
END_VAR

// Simulation variables
VAR
	EstopInput	: BOOL;
	LowAirInput : BOOL;
	ErrorInput	: BOOL;
	WarnInput	: BOOL;
	InfoInput	: BOOL;
END_VAR

//Need this FB to be RESET only to start safety comms ready for Safety Reset

//Available Safety FBS
//FB_Component_Safety_AndOrFB

METHOD PROTECTED Completing
VAR_INPUT
END_VAR
CASE _CurrentMode OF
	//=================================PRODUCTION MODE==================================
	E_PMLUnitMode.ePMLUnitMode_Production:
		StateComplete();

	E_PMLUnitMode.ePMLUnitMode_Maintenance, E_PMLUnitMode.ePMLUnitMode_Manual:
		SUPER^.Completing();
END_CASE
END_METHOD

METHOD PROTECTED CreateEvents
VAR_INPUT
END_VAR
// Add your event creation here
F_CreateAllEventsInClass(Alarms		:= MachineSafetyAlarms,
						 ClassSize	:= SIZEOF(TC_Events.DemoSystem),
						 pInitEvent := ADR(TC_EVENTS.DemoSystem.InitReferenceEvent),
						 Prefix		:= Name);

// Super call to base
SUPER^.CreateEvents();
END_METHOD

METHOD CyclicLogic
VAR_INPUT
END_VAR
IF NOT _InitComplete THEN
	_InitComplete := Initialize();
	RETURN;
END_IF

SUPER^.CyclicLogic();

// Fill in the PackTags for the machine output
_PackTags.Status.StateCurrent	 := _CurrentState;
_PackTags.Status.UnitModeCurrent := _CurrentMode;
UpdateModeTimers();


//Safety
//SafetyGroup_IO.CyclicLogic();
//SafetyGroup_ESTOP.CyclicLogic();

//This is just to simulate some IO for alarms
//CyclicLogic_Simulation();
END_METHOD

METHOD CyclicLogic_Simulation
VAR_INPUT
END_VAR

VAR_INST
END_VAR
(*	
This is just for testing. Real hardware can be setup in other places
Here the alarms will raise and clear on its own if the input changes	
*)
IF EstopInput AND NOT MachineAlarms[E_VFFSDemo.EmergencyStop].bRaised THEN
	RaiseAlarm2Args(MachineAlarms[E_VFFSDemo.EmergencyStop], '', '');
ELSIF NOT EstopInput AND MachineAlarms[E_VFFSDemo.EmergencyStop].bRaised THEN
	MachineAlarms[E_VFFSDemo.EmergencyStop].Clear(0, 0);
END_IF

IF LowAirInput AND NOT MachineAlarms[E_VFFSDemo.LowAir].bRaised THEN
	RaiseAlarm2Args(MachineAlarms[E_VFFSDemo.LowAir], '', '');
ELSIF NOT LowAirInput AND MachineAlarms[E_VFFSDemo.LowAir].bRaised THEN
	MachineAlarms[E_VFFSDemo.LowAir].Clear(0, 0);
END_IF

//Generic Alarms for Testing
IF ErrorInput AND NOT MachineAlarms[E_VFFSDemo.AlarmMessage].bRaised THEN
	RaiseAlarm2Args(MachineAlarms[E_VFFSDemo.AlarmMessage], '', '');
ELSIF NOT ErrorInput AND MachineAlarms[E_VFFSDemo.AlarmMessage].bRaised THEN
	MachineAlarms[E_VFFSDemo.AlarmMessage].Clear(0, 0);
END_IF

IF WarnInput AND NOT MachineAlarms[E_VFFSDemo.WarnMessage].bRaised THEN
	RaiseAlarm2Args(MachineAlarms[E_VFFSDemo.WarnMessage], '', '');
ELSIF NOT WarnInput AND MachineAlarms[E_VFFSDemo.WarnMessage].bRaised THEN
	MachineAlarms[E_VFFSDemo.WarnMessage].Clear(0, 0);
END_IF

IF InfoInput AND NOT MachineAlarms[E_VFFSDemo.InfoMessage].bRaised THEN
	RaiseAlarm2Args(MachineAlarms[E_VFFSDemo.InfoMessage], '', '');
ELSIF NOT InfoInput AND MachineAlarms[E_VFFSDemo.InfoMessage].bRaised THEN
	MachineAlarms[E_VFFSDemo.InfoMessage].Clear(0, 0);
END_IF
END_METHOD

METHOD PROTECTED FINAL Execute
VAR_INPUT
END_VAR
CASE _CurrentMode OF
	//=================================PRODUCTION MODE==================================
	E_PMLUnitMode.ePMLUnitMode_Production:
		(* Run the sequence to make products 
		 Unwind Runs Slowly 
		 Pull Wheels Run 
		 Jaws Seal, and Repeat until production reached*)
//		sealTrig(CLK := SequenceState = 10);
//		IF sealTrig.Q THEN
//			partTimeStart := F_GetActualDcTime64();
//			sealTimeStart := partTimeStart;
//		END_IF

//		pulltrig(CLK := SequenceState = 20);
//		IF pulltrig.Q THEN
//			pullTimeStart := F_GetActualDcTime64();
//		END_IF

//		IF THIS^.Sealer.sealbar.InTempRange THEN
//			CASE SequenceState OF
//				0: //Started
//					Unwind.ChangeState(E_PMLCommand.ePMLCommand_Start);
//					IF Unwind.CurrentState = E_PMLState.ePMLState_Execute THEN
//						SequenceState := SequenceState + 10;
//					END_IF

//				10: // SEAL First
//					Sealer.ChangeState(E_PMLCommand.ePMLCommand_Start);
//					IF Sealer.CurrentState = E_PMLState.ePMLState_Complete THEN
//						Sealer.ChangeState(E_PMLCommand.ePMLCommand_Reset);
//						SequenceState := SequenceState + 10;
//						SealTimeEnd	  := F_GetActualDcTime64();
//						sealingTime	  := ULINT_TO_LREAL(sealtimeEnd - sealTimeStart) * 1E-9;
//					END_IF

//				20: // Run Pullwheels
//					PullWheels.ChangeState(E_PMLCommand.ePMLCommand_Start);
//					IF PullWheels.CurrentState = E_PMLState.ePMLState_Complete THEN
//						partTimeEnd	  := F_GetActualDcTime64();
//						parts		  := parts + 1;
//						SequenceState := 10;
//						PullWheels.ChangeState(E_PMLCommand.ePMLCommand_Reset);
//						pullTimeEnd := F_GetActualDcTime64();
//						pullingTime := ULINT_TO_LREAL(pullTimeEnd - pullTimeStart) * 1E-9;
//					END_IF
//			END_CASE
//		ELSE
//			ChangeState(E_PMLCommand.ePMLCommand_Suspend);
//		END_IF

	//=================================MAINTENANCE MODE==================================	
	E_PMLUnitMode.ePMLUnitMode_Maintenance:
		;

	//=================================MANUAL MODE==================================
	E_PMLUnitMode.ePMLUnitMode_Manual:
		;
END_CASE
END_METHOD

METHOD PROTECTED Held
VAR_INPUT
END_VAR
END_METHOD

METHOD PROTECTED HMIPermissions
VAR_INPUT
END_VAR
//General Mode Based Monitoring and handling of HMI control
CASE _CurrentMode OF
	E_PMLUnitMode.ePMLUnitMode_Production:
		CASE _CurrentState OF
			E_PMLState.ePMLState_Stopped:
				AllowHMIControl(ThisModuleOnly := TRUE); //Allow control for recovery
			E_PMLState.ePMLState_Idle:
				//BlockHMIControl();
				AllowHMIControl(ThisModuleOnly := TRUE); //Allow control for recovery
			E_PMLState.ePMLState_Suspended:
				BlockHMIControl();

			E_PMLState.ePMLState_Execute:
				BlockHMIControl();

			E_PMLState.ePMLState_Aborted:
				AllowHMIControl(ThisModuleOnly := TRUE); //Allow control for recovery
			E_PMLState.ePMLState_Held:
				AllowHMIControl(ThisModuleOnly := TRUE); //Allow control for recovery
			E_PMLState.ePMLState_Complete:
				BlockHMIControl();
		END_CASE

	//AllowHMIControl(ThisModuleOnly := FALSE);
	E_PMLUnitMode.ePMLUnitMode_Manual:
		AllowHMIControl(ThisModuleOnly := FALSE);

	E_PMLUnitMode.ePMLUnitMode_Maintenance:
		AllowHMIControl(ThisModuleOnly := FALSE);
END_CASE
END_METHOD

METHOD PROTECTED HoldImmediate
VAR_INPUT
END_VAR
ChangeState(E_PMLCommand.ePMLCommand_Hold);
END_METHOD

METHOD PROTECTED Holding
VAR_INPUT
END_VAR
CASE _CurrentMode OF
	//=================================PRODUCTION MODE==================================
	E_PMLUnitMode.ePMLUnitMode_Production:
	//	IF (Sealer.CurrentState = E_PMLState.ePMLState_Complete OR Sealer.CurrentState = E_PMLState.ePMLState_Idle) AND (PullWheels.CurrentState = E_PMLState.ePMLState_Complete OR PullWheels.CurrentState = E_PMLState.ePMLState_Idle) THEN
			StateComplete();
	//	END_IF

	E_PMLUnitMode.ePMLUnitMode_Maintenance, E_PMLUnitMode.ePMLUnitMode_Manual:
		SUPER^.Holding();
END_CASE
END_METHOD

METHOD PROTECTED Initialize : BOOL
VAR
	i : UDINT; //Generic iteration value
END_VAR
Initialize := FALSE;
CASE DescendantSequenceState OF
	0:
		//Groups
		RegisterComponent(SafetyGroup_IO);
		RegisterComponent(SafetyGroup_ESTOP);
		RegisterComponent(SafetyOutput);
		RegisterComponent(SafetyInput);
		
		//Safety Circuit components
		RegisterComponent(Reset_PB);
		RegisterComponent(SafetyEstop);
		RegisterComponent(Safty_Reset_Pulse_Out);
		
		
		_LogModeChanges			:= FALSE;
		_LogStateChanges		:= FALSE;
		DescendantSequenceState := DescendantSequenceState + 10;

	10:
		//Setup Custom modes here

		CustomModes(eMode                          :=,
                    sName                          :='Safety Module_Mode',
                    bDisableClearing               :=TRUE,
                    bDisableStarting               :=,
                    bDisableSuspended              :=TRUE,
                    bDisableStopping               :=TRUE,
                    bDisableAborting               :=,
                    bDisableHolding                :=TRUE,
                    bDisableHeld                   :=TRUE,
                    bDisableUnholding              :=TRUE,
                    bDisableSuspending             :=TRUE,
                    bDisableUnsuspending           :=TRUE,
                    bDisableResetting              :=,
                    bDisableIdle                   :=TRUE,
                    bDisableCompleting             :=TRUE,
                    bDisableComplete               :=TRUE,
                    bEnableUnitModeChangeStopped   :=,
                    bEnableUnitModeChangeIdle      :=TRUE,
                    bEnableUnitModeChangeSuspended :=TRUE,
                    bEnableUnitModeChangeExecute   :=,
                    bEnableUnitModeChangeAborted   :=,
                    bEnableUnitModeChangeHeld      :=TRUE,
                    bEnableUnitModeChangeComplete  :=,
                    bError                         =>,
                    nErrorId                       =>);
		DescendantSequenceState := DescendantSequenceState + 10;

	20:
		//Copy Mode names
		FOR i := 1 TO 3 DO
			ModeNames[i] := F_UnitModeToString(UDINT_TO_DINT(i));
		END_FOR

		DescendantSequenceState := DescendantSequenceState + 10;

	30:
		// Initialize Recipes 
		Initialize_Recipes();
		DescendantSequenceState := DescendantSequenceState + 10;

	40:
		//Call the Super
		IF SUPER^.Initialize() THEN
			DescendantSequenceState := DescendantSequenceState + 10;
		END_IF

	50:
		Initialize := TRUE;
END_CASE
END_METHOD

METHOD Initialize_Recipes
VAR_INPUT
END_VAR
// configuration of parameters Max Speed
_packTags.Command.Parameter[1].ID	 := 1;
_packTags.Command.Parameter[1].Name	 := 'Max Speed';
_packTags.Command.Parameter[1].Unit	 := '/min';
_packTags.Command.Parameter[1].Value := 180;
_packTags.Command.Parameter[2].ID	 := 2;
_packTags.Command.Parameter[2].Name	 := 'Product to Run';
_packTags.Command.Parameter[2].Unit	 := '';
_packTags.Command.Parameter[2].Value := 1;

// Recipe Product 1
_PackTags.Command.Product[1].ProductID								:= 100;
_PackTags.Command.Product[1].Ingredients[1].IngredientID			:= 1;
_PackTags.Command.Product[1].Ingredients[1].Parameter[1].ID			:= _PackTags.Command.Product[1].ProductID * 10 + 1;
_PackTags.Command.Product[1].Ingredients[1].Parameter[1].Name		:= 'Material Type';
_PackTags.Command.Product[1].Ingredients[1].Parameter[1].Unit		:= 'n/a';
_PackTags.Command.Product[1].Ingredients[1].Parameter[1].Value		:= 5;
_PackTags.Command.Product[1].Ingredients[1].Parameter[2].ID			:= _PackTags.Command.Product[1].ProductID * 10 + 2;
_PackTags.Command.Product[1].Ingredients[1].Parameter[2].Name		:= 'Material Thickness';
_PackTags.Command.Product[1].Ingredients[1].Parameter[2].Unit		:= 'um';
_PackTags.Command.Product[1].Ingredients[1].Parameter[2].Value		:= 240;
_PackTags.Command.Product[1].ProcessVariables[LENGTH].ID			:= _PackTags.Command.Product[1].ProductID * 20 + 1;
_PackTags.Command.Product[1].ProcessVariables[LENGTH].Name			:= 'Length';
_PackTags.Command.Product[1].ProcessVariables[LENGTH].Unit			:= 'mm';
_PackTags.Command.Product[1].ProcessVariables[LENGTH].Value			:= 100;
_PackTags.Command.Product[1].ProcessVariables[SEALTEMP].ID			:= _PackTags.Command.Product[1].ProductID * 20 + 2;
_PackTags.Command.Product[1].ProcessVariables[SEALTEMP].Name		:= 'Sealing Temp';
_PackTags.Command.Product[1].ProcessVariables[SEALTEMP].Unit		:= 'C';
_PackTags.Command.Product[1].ProcessVariables[SEALTEMP].Value		:= 100;
_PackTags.Command.Product[1].ProcessVariables[SEALTIME].ID			:= _PackTags.Command.Product[1].ProductID * 20 + 3;
_PackTags.Command.Product[1].ProcessVariables[SEALTIME].Name		:= 'Sealing Time';
_PackTags.Command.Product[1].ProcessVariables[SEALTIME].Unit		:= 'ms';
_PackTags.Command.Product[1].ProcessVariables[SEALTIME].Value		:= 50;
_PackTags.Command.Product[1].ProcessVariables[PULLWHEELS_VEL].ID	:= _PackTags.Command.Product[1].ProductID * 20 + 4;
_PackTags.Command.Product[1].ProcessVariables[PULLWHEELS_VEL].Name	:= 'Pull Wheels Vel';
_PackTags.Command.Product[1].ProcessVariables[PULLWHEELS_VEL].Unit	:= 'mm/s';
_PackTags.Command.Product[1].ProcessVariables[PULLWHEELS_VEL].Value := 100;
_PackTags.Command.Product[1].ProcessVariables[PULLWHEELS_ACC].ID	:= _PackTags.Command.Product[1].ProductID * 20 + 5;
_PackTags.Command.Product[1].ProcessVariables[PULLWHEELS_ACC].Name	:= 'Pull Wheels Acc';
_PackTags.Command.Product[1].ProcessVariables[PULLWHEELS_ACC].Unit	:= 'mm/s2';
_PackTags.Command.Product[1].ProcessVariables[PULLWHEELS_ACC].Value := 1000;
_PackTags.Command.Product[1].ProcessVariables[OPEN_POS].ID			:= _PackTags.Command.Product[1].ProductID * 20 + 6;
_PackTags.Command.Product[1].ProcessVariables[OPEN_POS].Name		:= 'Sealer Open Position';
_PackTags.Command.Product[1].ProcessVariables[OPEN_POS].Unit		:= 'mm';
_PackTags.Command.Product[1].ProcessVariables[OPEN_POS].Value		:= 105;
_PackTags.Command.Product[1].ProcessVariables[CLOSED_POS].ID		:= _PackTags.Command.Product[1].ProductID * 20 + 7;
_PackTags.Command.Product[1].ProcessVariables[CLOSED_POS].Name		:= 'Sealer Closed Position';
_PackTags.Command.Product[1].ProcessVariables[CLOSED_POS].Unit		:= 'mm';
_PackTags.Command.Product[1].ProcessVariables[CLOSED_POS].Value		:= 250;
_PackTags.Command.Product[1].ProcessVariables[SEALER_VEL].ID		:= _PackTags.Command.Product[1].ProductID * 20 + 8;
_PackTags.Command.Product[1].ProcessVariables[SEALER_VEL].Name		:= 'Sealer Vel';
_PackTags.Command.Product[1].ProcessVariables[SEALER_VEL].Unit		:= 'mm/s';
_PackTags.Command.Product[1].ProcessVariables[SEALER_VEL].Value		:= 100;
_PackTags.Command.Product[1].ProcessVariables[SEALER_ACC].ID		:= _PackTags.Command.Product[1].ProductID * 20 + 9;
_PackTags.Command.Product[1].ProcessVariables[SEALER_ACC].Name		:= 'Sealer Acc';
_PackTags.Command.Product[1].ProcessVariables[SEALER_ACC].Unit		:= 'mm/s2';
_PackTags.Command.Product[1].ProcessVariables[SEALER_ACC].Value		:= 1000;
_PackTags.Command.Product[1].ProcessVariables[UNWIND_VEL].ID		:= _PackTags.Command.Product[1].ProductID * 20 + 10;
_PackTags.Command.Product[1].ProcessVariables[UNWIND_VEL].Name		:= 'Unwind Vel';
_PackTags.Command.Product[1].ProcessVariables[UNWIND_VEL].Unit		:= 'mm/s';
_PackTags.Command.Product[1].ProcessVariables[UNWIND_VEL].Value		:= 100;
_PackTags.Command.Product[1].ProcessVariables[UNWIND_ACC].ID		:= _PackTags.Command.Product[1].ProductID * 20 + 11;
_PackTags.Command.Product[1].ProcessVariables[UNWIND_ACC].Name		:= 'Unwind Acc';
_PackTags.Command.Product[1].ProcessVariables[UNWIND_ACC].Unit		:= 'mm/s2';
_PackTags.Command.Product[1].ProcessVariables[UNWIND_ACC].Value		:= 1000;

// Product 2
_PackTags.Command.Product[2].ProductID								:= 100;
_PackTags.Command.Product[2].Ingredients[1].IngredientID			:= 1;
_PackTags.Command.Product[2].Ingredients[1].Parameter[1].ID			:= _PackTags.Command.Product[1].ProductID * 10 + 1;
_PackTags.Command.Product[2].Ingredients[1].Parameter[1].Name		:= 'Material Type';
_PackTags.Command.Product[2].Ingredients[1].Parameter[1].Unit		:= 'n/a';
_PackTags.Command.Product[2].Ingredients[1].Parameter[1].Value		:= 2;
_PackTags.Command.Product[2].Ingredients[1].Parameter[2].ID			:= _PackTags.Command.Product[1].ProductID * 10 + 2;
_PackTags.Command.Product[2].Ingredients[1].Parameter[2].Name		:= 'Material Thickness';
_PackTags.Command.Product[2].Ingredients[1].Parameter[2].Unit		:= 'um';
_PackTags.Command.Product[2].Ingredients[1].Parameter[2].Value		:= 220;
_PackTags.Command.Product[2].ProcessVariables[LENGTH].ID			:= _PackTags.Command.Product[1].ProductID * 20 + 1;
_PackTags.Command.Product[2].ProcessVariables[LENGTH].Name			:= 'Length';
_PackTags.Command.Product[2].ProcessVariables[LENGTH].Unit			:= 'mm';
_PackTags.Command.Product[2].ProcessVariables[LENGTH].Value			:= 55;
_PackTags.Command.Product[2].ProcessVariables[SEALTEMP].ID			:= _PackTags.Command.Product[1].ProductID * 20 + 2;
_PackTags.Command.Product[2].ProcessVariables[SEALTEMP].Name		:= 'Sealing Temp';
_PackTags.Command.Product[2].ProcessVariables[SEALTEMP].Unit		:= 'C';
_PackTags.Command.Product[2].ProcessVariables[SEALTEMP].Value		:= 110;
_PackTags.Command.Product[2].ProcessVariables[SEALTIME].ID			:= _PackTags.Command.Product[1].ProductID * 20 + 3;
_PackTags.Command.Product[2].ProcessVariables[SEALTIME].Name		:= 'Sealing Time';
_PackTags.Command.Product[2].ProcessVariables[SEALTIME].Unit		:= 'ms';
_PackTags.Command.Product[2].ProcessVariables[SEALTIME].Value		:= 100;
_PackTags.Command.Product[2].ProcessVariables[PULLWHEELS_VEL].ID	:= _PackTags.Command.Product[1].ProductID * 20 + 4;
_PackTags.Command.Product[2].ProcessVariables[PULLWHEELS_VEL].Name	:= 'Pull Wheels Vel';
_PackTags.Command.Product[2].ProcessVariables[PULLWHEELS_VEL].Unit	:= 'mm/s';
_PackTags.Command.Product[2].ProcessVariables[PULLWHEELS_VEL].Value := 200;
_PackTags.Command.Product[2].ProcessVariables[PULLWHEELS_ACC].ID	:= _PackTags.Command.Product[1].ProductID * 20 + 5;
_PackTags.Command.Product[2].ProcessVariables[PULLWHEELS_ACC].Name	:= 'Pull Wheels Acc';
_PackTags.Command.Product[2].ProcessVariables[PULLWHEELS_ACC].Unit	:= 'mm/s2';
_PackTags.Command.Product[2].ProcessVariables[PULLWHEELS_ACC].Value := 2000;
_PackTags.Command.Product[2].ProcessVariables[OPEN_POS].ID			:= _PackTags.Command.Product[1].ProductID * 20 + 6;
_PackTags.Command.Product[2].ProcessVariables[OPEN_POS].Name		:= 'Sealer Open Position';
_PackTags.Command.Product[2].ProcessVariables[OPEN_POS].Unit		:= 'mm';
_PackTags.Command.Product[2].ProcessVariables[OPEN_POS].Value		:= 60;
_PackTags.Command.Product[2].ProcessVariables[CLOSED_POS].ID		:= _PackTags.Command.Product[1].ProductID * 20 + 7;
_PackTags.Command.Product[2].ProcessVariables[CLOSED_POS].Name		:= 'Sealer Closed Position';
_PackTags.Command.Product[2].ProcessVariables[CLOSED_POS].Unit		:= 'mm';
_PackTags.Command.Product[2].ProcessVariables[CLOSED_POS].Value		:= 253;
_PackTags.Command.Product[2].ProcessVariables[SEALER_VEL].ID		:= _PackTags.Command.Product[1].ProductID * 20 + 8;
_PackTags.Command.Product[2].ProcessVariables[SEALER_VEL].Name		:= 'Sealer Vel';
_PackTags.Command.Product[2].ProcessVariables[SEALER_VEL].Unit		:= 'mm/s';
_PackTags.Command.Product[2].ProcessVariables[SEALER_VEL].Value		:= 200;
_PackTags.Command.Product[2].ProcessVariables[SEALER_ACC].ID		:= _PackTags.Command.Product[1].ProductID * 20 + 9;
_PackTags.Command.Product[2].ProcessVariables[SEALER_ACC].Name		:= 'Sealer Acc';
_PackTags.Command.Product[2].ProcessVariables[SEALER_ACC].Unit		:= 'mm/s2';
_PackTags.Command.Product[2].ProcessVariables[SEALER_ACC].Value		:= 2000;
_PackTags.Command.Product[2].ProcessVariables[UNWIND_VEL].ID		:= _PackTags.Command.Product[1].ProductID * 20 + 10;
_PackTags.Command.Product[2].ProcessVariables[UNWIND_VEL].Name		:= 'Unwind Vel';
_PackTags.Command.Product[2].ProcessVariables[UNWIND_VEL].Unit		:= 'mm/s';
_PackTags.Command.Product[2].ProcessVariables[UNWIND_VEL].Value		:= 200;
_PackTags.Command.Product[2].ProcessVariables[UNWIND_ACC].ID		:= _PackTags.Command.Product[1].ProductID * 20 + 11;
_PackTags.Command.Product[2].ProcessVariables[UNWIND_ACC].Name		:= 'Unwind Acc';
_PackTags.Command.Product[2].ProcessVariables[UNWIND_ACC].Unit		:= 'mm/s2';
_PackTags.Command.Product[2].ProcessVariables[UNWIND_ACC].Value		:= 2000;

